KUKA KRL program: f1_Kuka_APT223T02S23.SRC

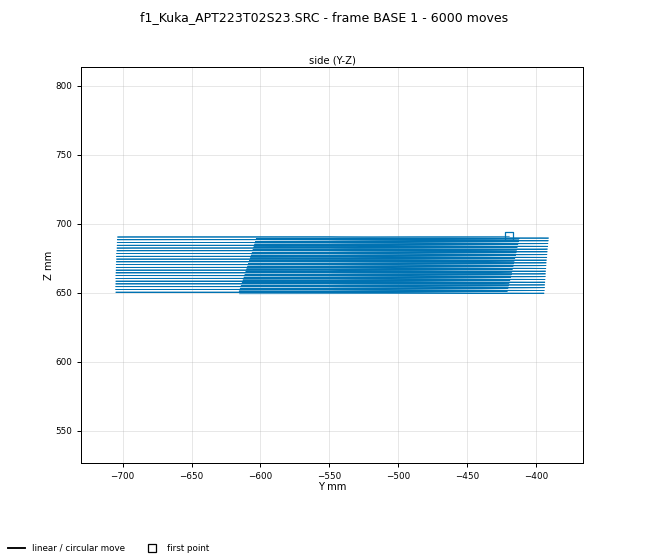
[picture p0: tool path of f1_Kuka_APT223T02S23.SRC in frame BASE 1, 6000 of 6001 moves have a stored position in this frame; points joined in program order, loops and branches not executed]
&ACCESS RVP
&REL 2
&PARAM TEMPLATE = C:\KRC\Roboter\Template\vorgabe
&PARAM EDITMASK = *
DEF f1_Kuka_APT223T02S23()


;FOLD INI;%{PE}%V3.2.0,%MKUKATPBASIS,%CINIT,%VCOMMON,%P
  ;FOLD BAS INI;%{E}%V3.2.0,%MKUKATPBASIS,%CINIT,%VINIT,%P
    GLOBAL INTERRUPT DECL 3 WHEN $STOPMESS==TRUE DO IR_STOPM ( )
    INTERRUPT ON 3
    BAS (#INITMOV,0 )
  ;ENDFOLD (BAS INI)
  ;FOLD USER INI;%{E}%V3.2.0,%MKUKATPUSER,%CINIT,%VINIT,%P
    ;Make your modifications here
  ;ENDFOLD (USER INI)
;ENDFOLD (INI)


;*** Make Null PTP Move
  PTP $pos_act

;*** Auto Load The Correct TOOL Data
  $tool=tool_data[2]

;*** Auto Load The Correct BASE Data
  $base=base_data[1]

  $ADVANCE = 5

;*** Restate Last Velocity
MMPM(30000.0)
SetRPM(8000)
LIN {X -0.177,Y -419.662,Z 690.937,A 0.000,B 0.000,C 90.000,E1 24.591} C_DIS
LIN {X 0.038,Y -422.624,Z 690.918,A 0.000,B 0.000,C 90.000,E1 21.173} C_DIS
LIN {X -0.096,Y -424.250,Z 690.908,A 0.000,B 0.000,C 90.000,E1 19.504} C_DIS
LIN {X -0.088,Y -425.859,Z 690.899,A 0.000,B 0.000,C 90.000,E1 17.819} C_DIS
LIN {X 0.034,Y -427.863,Z 690.888,A 0.000,B 0.000,C 90.000,E1 15.788} C_DIS
LIN {X -0.122,Y -430.468,Z 690.875,A 0.000,B 0.000,C 90.000,E1 13.467} C_DIS
LIN {X 0.099,Y -432.415,Z 690.866,A 0.000,B 0.000,C 90.000,E1 11.771} C_DIS
LIN {X -0.143,Y -434.451,Z 690.856,A 0.000,B 0.000,C 90.000,E1 10.141} C_DIS
LIN {X -0.149,Y -438.666,Z 690.838,A 0.000,B 0.000,C 90.000,E1 6.834} C_DIS
LIN {X -0.142,Y -441.750,Z 690.825,A 0.000,B 0.000,C 90.000,E1 4.531} C_DIS
LIN {X 0.024,Y -445.734,Z 690.811,A 0.000,B 0.000,C 90.000,E1 1.892} C_DIS
LIN {X -0.126,Y -449.793,Z 690.797,A 0.000,B 0.000,C 90.000,E1 359.484} C_DIS
LIN {X -0.170,Y -454.545,Z 690.783,A 0.000,B 0.000,C 90.000,E1 356.906} C_DIS
LIN {X 0.066,Y -458.306,Z 690.772,A 0.000,B 0.000,C 90.000,E1 354.951} C_DIS
LIN {X 0.178,Y -462.682,Z 690.760,A 0.000,B 0.000,C 90.000,E1 352.704} C_DIS
LIN {X -0.197,Y -466.311,Z 690.749,A 0.000,B 0.000,C 90.000,E1 350.849} C_DIS
LIN {X 0.236,Y -469.219,Z 690.740,A 0.000,B 0.000,C 90.000,E1 349.218} C_DIS
LIN {X 0.085,Y -472.585,Z 690.730,A 0.000,B 0.000,C 90.000,E1 347.353} C_DIS
LIN {X 0.213,Y -475.984,Z 690.719,A 0.000,B 0.000,C 90.000,E1 345.463} C_DIS
LIN {X 0.089,Y -479.488,Z 690.709,A 0.000,B 0.000,C 90.000,E1 343.614} C_DIS
LIN {X 0.195,Y -482.545,Z 690.701,A 0.000,B 0.000,C 90.000,E1 342.054} C_DIS
LIN {X 0.039,Y -484.409,Z 690.695,A 0.000,B 0.000,C 90.000,E1 341.148} C_DIS
LIN {X -0.067,Y -487.532,Z 690.687,A 0.000,B 0.000,C 90.000,E1 339.625} C_DIS
LIN {X -0.060,Y -491.876,Z 690.675,A 0.000,B 0.000,C 90.000,E1 337.486} C_DIS
LIN {X 0.051,Y -493.742,Z 690.670,A 0.000,B 0.000,C 90.000,E1 336.561} C_DIS
LIN {X -0.118,Y -495.162,Z 690.667,A 0.000,B 0.000,C 90.000,E1 335.973} C_DIS
LIN {X -0.024,Y -496.658,Z 690.663,A 0.000,B 0.000,C 90.000,E1 335.357} C_DIS
LIN {X -0.171,Y -498.186,Z 690.661,A 0.000,B 0.000,C 90.000,E1 334.921} C_DIS
LIN {X 0.097,Y -499.596,Z 690.659,A 0.000,B 0.000,C 90.000,E1 334.588} C_DIS
LIN {X -0.042,Y -501.612,Z 690.657,A 0.000,B 0.000,C 90.000,E1 334.280} C_DIS
LIN {X 0.069,Y -505.458,Z 690.655,A 0.000,B 0.000,C 90.000,E1 333.819} C_DIS
LIN {X -0.161,Y -510.103,Z 690.652,A 0.000,B 0.000,C 90.000,E1 333.435} C_DIS
LIN {X -0.285,Y -521.797,Z 690.648,A 0.000,B 0.000,C 90.000,E1 332.615} C_DIS
LIN {X -0.135,Y -531.169,Z 690.644,A 0.000,B 0.000,C 90.000,E1 331.975} C_DIS
LIN {X 0.252,Y -537.247,Z 690.642,A 0.000,B 0.000,C 90.000,E1 331.513} C_DIS
LIN {X 0.307,Y -541.703,Z 690.640,A 0.000,B 0.000,C 90.000,E1 331.179} C_DIS
LIN {X 0.113,Y -547.474,Z 690.638,A 0.000,B 0.000,C 90.000,E1 330.745} C_DIS
LIN {X 0.018,Y -553.101,Z 690.635,A 0.000,B 0.000,C 90.000,E1 330.284} C_DIS
LIN {X 0.032,Y -561.262,Z 690.631,A 0.000,B 0.000,C 90.000,E1 329.537} C_DIS
LIN {X -0.119,Y -571.528,Z 690.625,A 0.000,B 0.000,C 90.000,E1 328.535} C_DIS
LIN {X 0.210,Y -580.334,Z 690.620,A 0.000,B 0.000,C 90.000,E1 327.582} C_DIS
LIN {X -0.169,Y -591.315,Z 690.613,A 0.000,B 0.000,C 90.000,E1 326.421} C_DIS
LIN {X 0.068,Y -600.742,Z 690.608,A 0.000,B 0.000,C 90.000,E1 325.341} C_DIS
LIN {X 0.066,Y -605.196,Z 690.605,A 0.000,B 0.000,C 90.000,E1 324.815} C_DIS
LIN {X -0.294,Y -610.378,Z 690.601,A 0.000,B 0.000,C 90.000,E1 324.196} C_DIS
LIN {X 0.048,Y -617.140,Z 690.596,A 0.000,B 0.000,C 90.000,E1 323.256} C_DIS
LIN {X -0.223,Y -621.759,Z 690.592,A 0.000,B 0.000,C 90.000,E1 322.637} C_DIS
LIN {X 0.114,Y -629.358,Z 690.586,A 0.000,B 0.000,C 90.000,E1 321.457} C_DIS
LIN {X 0.322,Y -633.342,Z 690.582,A 0.000,B 0.000,C 90.000,E1 320.803} C_DIS
LIN {X 0.059,Y -637.842,Z 690.578,A 0.000,B 0.000,C 90.000,E1 320.070} C_DIS
LIN {X 0.157,Y -644.321,Z 690.572,A 0.000,B 0.000,C 90.000,E1 318.933} C_DIS
LIN {X 0.004,Y -647.101,Z 690.569,A 0.000,B 0.000,C 90.000,E1 318.447} C_DIS
LIN {X 0.242,Y -653.083,Z 690.563,A 0.000,B 0.000,C 90.000,E1 317.310} C_DIS
LIN {X 0.118,Y -656.784,Z 690.559,A 0.000,B 0.000,C 90.000,E1 316.581} C_DIS
LIN {X -0.428,Y -660.278,Z 690.555,A 0.000,B 0.000,C 90.000,E1 315.891} C_DIS
LIN {X -0.019,Y -663.506,Z 690.551,A 0.000,B 0.000,C 90.000,E1 315.121} C_DIS
LIN {X 0.423,Y -667.564,Z 690.545,A 0.000,B 0.000,C 90.000,E1 314.109} C_DIS
LIN {X -0.017,Y -671.440,Z 690.540,A 0.000,B 0.000,C 90.000,E1 313.176} C_DIS
LIN {X 0.069,Y -676.276,Z 690.533,A 0.000,B 0.000,C 90.000,E1 311.962} C_DIS
LIN {X -0.173,Y -680.748,Z 690.527,A 0.000,B 0.000,C 90.000,E1 310.782} C_DIS
LIN {X 0.106,Y -684.621,Z 690.520,A 0.000,B 0.000,C 90.000,E1 309.564} C_DIS
LIN {X 0.339,Y -686.758,Z 690.516,A 0.000,B 0.000,C 90.000,E1 308.830} C_DIS
LIN {X 0.221,Y -689.226,Z 690.511,A 0.000,B 0.000,C 90.000,E1 307.890} C_DIS
LIN {X 0.135,Y -691.500,Z 690.505,A 0.000,B 0.000,C 90.000,E1 306.950} C_DIS
LIN {X 0.073,Y -693.483,Z 690.500,A 0.000,B 0.000,C 90.000,E1 306.011} C_DIS
LIN {X -0.023,Y -694.830,Z 690.496,A 0.000,B 0.000,C 90.000,E1 305.311} C_DIS
LIN {X 0.245,Y -695.690,Z 690.494,A 0.000,B 0.000,C 90.000,E1 304.818} C_DIS
LIN {X -0.176,Y -697.121,Z 690.488,A 0.000,B 0.000,C 90.000,E1 303.913} C_DIS
LIN {X 0.344,Y -698.059,Z 690.484,A 0.000,B 0.000,C 90.000,E1 303.166} C_DIS
LIN {X -0.056,Y -699.136,Z 690.479,A 0.000,B 0.000,C 90.000,E1 302.260} C_DIS
LIN {X 0.061,Y -700.597,Z 690.471,A 0.000,B 0.000,C 90.000,E1 300.846} C_DIS
LIN {X 0.253,Y -701.115,Z 690.468,A 0.000,B 0.000,C 90.000,E1 300.129} C_DIS
LIN {X 0.050,Y -701.883,Z 690.460,A 0.000,B 0.000,C 90.000,E1 298.743} C_DIS
LIN {X 0.148,Y -702.599,Z 690.452,A 0.000,B 0.000,C 90.000,E1 297.334} C_DIS
LIN {X -0.078,Y -703.675,Z 690.443,A 0.000,B 0.000,C 90.000,E1 295.720} C_DIS
LIN {X -0.164,Y -703.404,Z 690.439,A 0.000,B 0.000,C 90.000,E1 295.027} C_DIS
LIN {X 0.399,Y -702.194,Z 690.436,A 0.000,B 0.000,C 90.000,E1 294.515} C_DIS
LIN {X -0.251,Y -701.369,Z 690.435,A 0.000,B 0.000,C 90.000,E1 294.335} C_DIS
LIN {X -0.113,Y -700.580,Z 690.435,A 0.000,B 0.000,C 90.000,E1 294.207} C_DIS
LIN {X 0.144,Y -696.444,Z 690.432,A 0.000,B 0.000,C 90.000,E1 293.718} C_DIS
LIN {X -0.363,Y -695.033,Z 690.431,A 0.000,B 0.000,C 90.000,E1 293.643} C_DIS
LIN {X -0.119,Y -692.958,Z 690.431,A 0.000,B 0.000,C 90.000,E1 293.515} C_DIS
LIN {X -0.070,Y -688.688,Z 690.430,A 0.000,B 0.000,C 90.000,E1 293.334} C_DIS
LIN {X -0.001,Y -684.521,Z 690.429,A 0.000,B 0.000,C 90.000,E1 293.206} C_DIS
LIN {X -0.212,Y -680.088,Z 690.428,A 0.000,B 0.000,C 90.000,E1 293.131} C_DIS
LIN {X 0.206,Y -675.238,Z 690.428,A 0.000,B 0.000,C 90.000,E1 293.025} C_DIS
LIN {X -0.219,Y -661.690,Z 690.427,A 0.000,B 0.000,C 90.000,E1 292.898} C_DIS
LIN {X -0.319,Y -644.942,Z 690.426,A 0.000,B 0.000,C 90.000,E1 292.642} C_DIS
LIN {X 0.098,Y -635.046,Z 690.425,A 0.000,B 0.000,C 90.000,E1 292.408} C_DIS
LIN {X 0.208,Y -621.578,Z 690.423,A 0.000,B 0.000,C 90.000,E1 292.078} C_DIS
LIN {X 0.164,Y -608.109,Z 690.421,A 0.000,B 0.000,C 90.000,E1 291.716} C_DIS
LIN {X -0.104,Y -576.806,Z 690.415,A 0.000,B 0.000,C 90.000,E1 290.791} C_DIS
LIN {X -0.048,Y -562.877,Z 690.413,A 0.000,B 0.000,C 90.000,E1 290.375} C_DIS
LIN {X -0.135,Y -558.097,Z 690.412,A 0.000,B 0.000,C 90.000,E1 290.174} C_DIS
LIN {X 0.037,Y -557.476,Z 690.412,A 0.000,B 0.000,C 90.000,E1 290.120} C_DIS
LIN {X -0.045,Y -555.543,Z 690.411,A 0.000,B 0.000,C 90.000,E1 289.939} C_DIS
LIN {X -0.085,Y -555.513,Z 690.411,A 0.000,B 0.000,C 90.000,E1 289.939} C_DIS
LIN {X -0.138,Y -554.733,Z 690.409,A 0.000,B 0.000,C 90.000,E1 289.631} C_DIS
LIN {X -0.156,Y -554.284,Z 690.407,A 0.000,B 0.000,C 90.000,E1 289.214} C_DIS
LIN {X 0.121,Y -553.763,Z 690.397,A 0.000,B 0.000,C 90.000,E1 287.511} C_DIS
LIN {X -0.066,Y -553.275,Z 690.390,A 0.000,B 0.000,C 90.000,E1 286.134} C_DIS
LIN {X 0.007,Y -552.908,Z 690.383,A 0.000,B 0.000,C 90.000,E1 285.009} C_DIS
LIN {X 0.194,Y -552.348,Z 690.376,A 0.000,B 0.000,C 90.000,E1 283.592} C_DIS
LIN {X -0.172,Y -551.606,Z 690.366,A 0.000,B 0.000,C 90.000,E1 281.951} C_DIS
LIN {X 0.098,Y -550.681,Z 690.355,A 0.000,B 0.000,C 90.000,E1 279.962} C_DIS
LIN {X -0.181,Y -549.760,Z 690.341,A 0.000,B 0.000,C 90.000,E1 277.466} C_DIS
LIN {X -0.056,Y -549.171,Z 690.326,A 0.000,B 0.000,C 90.000,E1 274.645} C_DIS
LIN {X 0.215,Y -549.047,Z 690.318,A 0.000,B 0.000,C 90.000,E1 273.212} C_DIS
LIN {X -0.105,Y -548.798,Z 690.312,A 0.000,B 0.000,C 90.000,E1 272.121} C_DIS
LIN {X 0.113,Y -548.447,Z 690.306,A 0.000,B 0.000,C 90.000,E1 270.974} C_DIS
LIN {X 0.263,Y -548.002,Z 690.301,A 0.000,B 0.000,C 90.000,E1 270.115} C_DIS
LIN {X -0.001,Y -547.042,Z 690.291,A 0.000,B 0.000,C 90.000,E1 268.453} C_DIS
LIN {X -0.210,Y -545.831,Z 690.281,A 0.000,B 0.000,C 90.000,E1 266.502} C_DIS
LIN {X 0.064,Y -544.611,Z 690.271,A 0.000,B 0.000,C 90.000,E1 264.780} C_DIS
LIN {X -0.203,Y -543.514,Z 690.263,A 0.000,B 0.000,C 90.000,E1 263.394} C_DIS
LIN {X 0.130,Y -541.476,Z 690.252,A 0.000,B 0.000,C 90.000,E1 261.376} C_DIS
LIN {X 0.172,Y -539.073,Z 690.238,A 0.000,B 0.000,C 90.000,E1 258.814} C_DIS
LIN {X -0.080,Y -538.081,Z 690.232,A 0.000,B 0.000,C 90.000,E1 257.701} C_DIS
LIN {X -0.160,Y -536.881,Z 690.224,A 0.000,B 0.000,C 90.000,E1 256.284} C_DIS
LIN {X 0.260,Y -535.598,Z 690.216,A 0.000,B 0.000,C 90.000,E1 254.810} C_DIS
LIN {X 0.273,Y -534.122,Z 690.208,A 0.000,B 0.000,C 90.000,E1 253.378} C_DIS
LIN {X -0.251,Y -532.665,Z 690.200,A 0.000,B 0.000,C 90.000,E1 252.000} C_DIS
LIN {X 0.059,Y -530.980,Z 690.190,A 0.000,B 0.000,C 90.000,E1 250.242} C_DIS
LIN {X -0.051,Y -529.919,Z 690.186,A 0.000,B 0.000,C 90.000,E1 249.390} C_DIS
LIN {X 0.057,Y -527.109,Z 690.174,A 0.000,B 0.000,C 90.000,E1 247.358} C_DIS
LIN {X -0.213,Y -525.432,Z 690.168,A 0.000,B 0.000,C 90.000,E1 246.230} C_DIS
LIN {X 0.033,Y -522.500,Z 690.158,A 0.000,B 0.000,C 90.000,E1 244.460} C_DIS
LIN {X 0.014,Y -520.939,Z 690.153,A 0.000,B 0.000,C 90.000,E1 243.589} C_DIS
LIN {X 0.112,Y -518.673,Z 690.147,A 0.000,B 0.000,C 90.000,E1 242.410} C_DIS
LIN {X -0.147,Y -515.816,Z 690.139,A 0.000,B 0.000,C 90.000,E1 240.973} C_DIS
LIN {X -0.023,Y -513.973,Z 690.134,A 0.000,B 0.000,C 90.000,E1 240.078} C_DIS
LIN {X -0.217,Y -510.196,Z 690.124,A 0.000,B 0.000,C 90.000,E1 238.329} C_DIS
LIN {X -0.114,Y -506.987,Z 690.116,A 0.000,B 0.000,C 90.000,E1 236.834} C_DIS
LIN {X 0.313,Y -504.278,Z 690.109,A 0.000,B 0.000,C 90.000,E1 235.595} C_DIS
LIN {X 0.168,Y -500.836,Z 690.101,A 0.000,B 0.000,C 90.000,E1 234.116} C_DIS
LIN {X 0.084,Y -497.917,Z 690.094,A 0.000,B 0.000,C 90.000,E1 232.924} C_DIS
LIN {X -0.138,Y -494.899,Z 690.087,A 0.000,B 0.000,C 90.000,E1 231.743} C_DIS
LIN {X -0.008,Y -490.504,Z 690.077,A 0.000,B 0.000,C 90.000,E1 229.908} C_DIS
LIN {X -0.075,Y -484.730,Z 690.064,A 0.000,B 0.000,C 90.000,E1 227.472} C_DIS
LIN {X -0.011,Y -479.137,Z 690.050,A 0.000,B 0.000,C 90.000,E1 225.000} C_DIS
LIN {X -0.104,Y -475.497,Z 690.041,A 0.000,B 0.000,C 90.000,E1 223.461} C_DIS
LIN {X -0.072,Y -470.576,Z 690.029,A 0.000,B 0.000,C 90.000,E1 221.272} C_DIS
LIN {X -0.258,Y -467.231,Z 690.021,A 0.000,B 0.000,C 90.000,E1 219.725} C_DIS
LIN {X 0.155,Y -463.901,Z 690.012,A 0.000,B 0.000,C 90.000,E1 218.096} C_DIS
LIN {X 0.034,Y -457.033,Z 689.992,A 0.000,B 0.000,C 90.000,E1 214.612} C_DIS
LIN {X -0.296,Y -454.541,Z 689.985,A 0.000,B 0.000,C 90.000,E1 213.372} C_DIS
LIN {X 0.140,Y -450.873,Z 689.974,A 0.000,B 0.000,C 90.000,E1 211.386} C_DIS
LIN {X -0.134,Y -446.600,Z 689.962,A 0.000,B 0.000,C 90.000,E1 209.155} C_DIS
LIN {X 0.027,Y -443.112,Z 689.951,A 0.000,B 0.000,C 90.000,E1 207.180} C_DIS
LIN {X 0.083,Y -439.517,Z 689.940,A 0.000,B 0.000,C 90.000,E1 205.207} C_DIS
LIN {X 0.027,Y -437.117,Z 689.933,A 0.000,B 0.000,C 90.000,E1 203.898} C_DIS
LIN {X 0.162,Y -433.497,Z 689.922,A 0.000,B 0.000,C 90.000,E1 201.897} C_DIS
LIN {X 0.072,Y -430.490,Z 689.913,A 0.000,B 0.000,C 90.000,E1 200.248} C_DIS
LIN {X 0.126,Y -426.762,Z 689.901,A 0.000,B 0.000,C 90.000,E1 198.236} C_DIS
LIN {X 0.010,Y -422.649,Z 689.888,A 0.000,B 0.000,C 90.000,E1 195.898} C_DIS
LIN {X 0.147,Y -419.745,Z 689.879,A 0.000,B 0.000,C 90.000,E1 194.189} C_DIS
LIN {X 0.069,Y -415.050,Z 689.864,A 0.000,B 0.000,C 90.000,E1 191.478} C_DIS
LIN {X -0.068,Y -411.729,Z 689.852,A 0.000,B 0.000,C 90.000,E1 189.443} C_DIS
LIN {X 0.094,Y -409.036,Z 689.843,A 0.000,B 0.000,C 90.000,E1 187.701} C_DIS
LIN {X 0.135,Y -406.468,Z 689.833,A 0.000,B 0.000,C 90.000,E1 185.967} C_DIS
LIN {X 0.002,Y -403.075,Z 689.820,A 0.000,B 0.000,C 90.000,E1 183.555} C_DIS
LIN {X 0.159,Y -400.088,Z 689.806,A 0.000,B 0.000,C 90.000,E1 181.088} C_DIS
LIN {X 0.110,Y -396.926,Z 689.789,A 0.000,B 0.000,C 90.000,E1 177.936} C_DIS
LIN {X 0.061,Y -394.730,Z 689.773,A 0.000,B 0.000,C 90.000,E1 175.122} C_DIS
LIN {X -0.117,Y -392.750,Z 689.751,A 0.000,B 0.000,C 90.000,E1 171.254} C_DIS
LIN {X -0.029,Y -392.123,Z 689.738,A 0.000,B 0.000,C 90.000,E1 168.757} C_DIS
LIN {X -0.101,Y -391.771,Z 689.728,A 0.000,B 0.000,C 90.000,E1 166.992} C_DIS
LIN {X -0.064,Y -391.172,Z 689.708,A 0.000,B 0.000,C 90.000,E1 163.433} C_DIS
LIN {X 0.188,Y -391.169,Z 689.692,A 0.000,B 0.000,C 90.000,E1 160.550} C_DIS
LIN {X 0.091,Y -391.330,Z 689.676,A 0.000,B 0.000,C 90.000,E1 157.720} C_DIS
LIN {X -0.089,Y -391.469,Z 689.664,A 0.000,B 0.000,C 90.000,E1 155.613} C_DIS
LIN {X -0.106,Y -391.736,Z 689.651,A 0.000,B 0.000,C 90.000,E1 153.127} C_DIS
LIN {X 0.105,Y -392.346,Z 689.635,A 0.000,B 0.000,C 90.000,E1 150.255} C_DIS
LIN {X -0.010,Y -393.124,Z 689.621,A 0.000,B 0.000,C 90.000,E1 147.788} C_DIS
LIN {X -0.212,Y -394.831,Z 689.601,A 0.000,B 0.000,C 90.000,E1 144.276} C_DIS
LIN {X 0.012,Y -396.062,Z 689.592,A 0.000,B 0.000,C 90.000,E1 142.477} C_DIS
LIN {X 0.158,Y -398.083,Z 689.578,A 0.000,B 0.000,C 90.000,E1 139.989} C_DIS
LIN {X 0.086,Y -399.704,Z 689.568,A 0.000,B 0.000,C 90.000,E1 138.243} C_DIS
LIN {X -0.047,Y -402.173,Z 689.555,A 0.000,B 0.000,C 90.000,E1 135.810} C_DIS
LIN {X 0.082,Y -403.736,Z 689.550,A 0.000,B 0.000,C 90.000,E1 134.919} C_DIS
LIN {X 0.078,Y -405.791,Z 689.546,A 0.000,B 0.000,C 90.000,E1 134.190} C_DIS
LIN {X -0.089,Y -407.601,Z 689.544,A 0.000,B 0.000,C 90.000,E1 133.866} C_DIS
LIN {X -0.210,Y -408.808,Z 689.542,A 0.000,B 0.000,C 90.000,E1 133.623} C_DIS
LIN {X -0.029,Y -410.740,Z 689.541,A 0.000,B 0.000,C 90.000,E1 133.338} C_DIS
LIN {X -0.106,Y -411.886,Z 689.540,A 0.000,B 0.000,C 90.000,E1 133.176} C_DIS
LIN {X -0.197,Y -416.632,Z 689.537,A 0.000,B 0.000,C 90.000,E1 132.690} C_DIS
LIN {X -0.118,Y -433.549,Z 689.529,A 0.000,B 0.000,C 90.000,E1 131.148} C_DIS
LIN {X 0.013,Y -448.902,Z 689.521,A 0.000,B 0.000,C 90.000,E1 129.850} C_DIS
LIN {X -0.164,Y -462.908,Z 689.515,A 0.000,B 0.000,C 90.000,E1 128.749} C_DIS
LIN {X 0.034,Y -468.842,Z 689.512,A 0.000,B 0.000,C 90.000,E1 128.222} C_DIS
LIN {X 0.051,Y -477.755,Z 689.508,A 0.000,B 0.000,C 90.000,E1 127.443} C_DIS
LIN {X -0.050,Y -484.911,Z 689.504,A 0.000,B 0.000,C 90.000,E1 126.790} C_DIS
LIN {X 0.072,Y -493.460,Z 689.500,A 0.000,B 0.000,C 90.000,E1 125.964} C_DIS
LIN {X -0.144,Y -498.944,Z 689.497,A 0.000,B 0.000,C 90.000,E1 125.438} C_DIS
LIN {X -0.289,Y -504.315,Z 689.494,A 0.000,B 0.000,C 90.000,E1 124.898} C_DIS
LIN {X -0.281,Y -507.046,Z 689.492,A 0.000,B 0.000,C 90.000,E1 124.612} C_DIS
LIN {X -0.129,Y -513.089,Z 689.488,A 0.000,B 0.000,C 90.000,E1 123.913} C_DIS
LIN {X -0.188,Y -516.672,Z 689.486,A 0.000,B 0.000,C 90.000,E1 123.499} C_DIS
LIN {X -0.176,Y -521.024,Z 689.483,A 0.000,B 0.000,C 90.000,E1 122.959} C_DIS
LIN {X -0.188,Y -525.187,Z 689.480,A 0.000,B 0.000,C 90.000,E1 122.418} C_DIS
LIN {X 0.169,Y -529.277,Z 689.477,A 0.000,B 0.000,C 90.000,E1 121.799} C_DIS
LIN {X 0.035,Y -533.666,Z 689.473,A 0.000,B 0.000,C 90.000,E1 121.131} C_DIS
LIN {X -0.162,Y -537.023,Z 689.470,A 0.000,B 0.000,C 90.000,E1 120.590} C_DIS
LIN {X -0.260,Y -541.499,Z 689.465,A 0.000,B 0.000,C 90.000,E1 119.745} C_DIS
LIN {X 0.085,Y -544.958,Z 689.461,A 0.000,B 0.000,C 90.000,E1 118.999} C_DIS
LIN {X 0.075,Y -548.802,Z 689.456,A 0.000,B 0.000,C 90.000,E1 118.153} C_DIS
LIN {X 0.083,Y -551.249,Z 689.453,A 0.000,B 0.000,C 90.000,E1 117.590} C_DIS
LIN {X 0.139,Y -554.580,Z 689.449,A 0.000,B 0.000,C 90.000,E1 116.744} C_DIS
LIN {X 0.006,Y -558.705,Z 689.443,A 0.000,B 0.000,C 90.000,E1 115.643} C_DIS
LIN {X -0.115,Y -561.579,Z 689.438,A 0.000,B 0.000,C 90.000,E1 114.823} C_DIS
LIN {X 0.309,Y -564.176,Z 689.433,A 0.000,B 0.000,C 90.000,E1 113.951} C_DIS
LIN {X 0.024,Y -566.557,Z 689.429,A 0.000,B 0.000,C 90.000,E1 113.153} C_DIS
LIN {X -0.014,Y -568.549,Z 689.424,A 0.000,B 0.000,C 90.000,E1 112.333} C_DIS
LIN {X -0.081,Y -571.418,Z 689.417,A 0.000,B 0.000,C 90.000,E1 110.972} C_DIS
LIN {X 0.247,Y -572.998,Z 689.412,A 0.000,B 0.000,C 90.000,E1 110.120} C_DIS
LIN {X -0.313,Y -575.878,Z 689.403,A 0.000,B 0.000,C 90.000,E1 108.544} C_DIS
LIN {X 0.078,Y -578.303,Z 689.395,A 0.000,B 0.000,C 90.000,E1 107.149} C_DIS
LIN {X 0.176,Y -580.646,Z 689.388,A 0.000,B 0.000,C 90.000,E1 105.788} C_DIS
LIN {X 0.098,Y -582.456,Z 689.382,A 0.000,B 0.000,C 90.000,E1 104.717} C_DIS
LIN {X 0.276,Y -584.612,Z 689.374,A 0.000,B 0.000,C 90.000,E1 103.355} C_DIS
LIN {X 0.034,Y -587.176,Z 689.365,A 0.000,B 0.000,C 90.000,E1 101.771} C_DIS
LIN {X -0.105,Y -588.958,Z 689.359,A 0.000,B 0.000,C 90.000,E1 100.715} C_DIS
LIN {X -0.067,Y -591.044,Z 689.352,A 0.000,B 0.000,C 90.000,E1 99.378} C_DIS
LIN {X 0.319,Y -592.602,Z 689.346,A 0.000,B 0.000,C 90.000,E1 98.276} C_DIS
LIN {X -0.059,Y -594.789,Z 689.337,A 0.000,B 0.000,C 90.000,E1 96.720} C_DIS
LIN {X 0.205,Y -596.779,Z 689.329,A 0.000,B 0.000,C 90.000,E1 95.106} C_DIS
LIN {X 0.227,Y -598.397,Z 689.321,A 0.000,B 0.000,C 90.000,E1 93.784} C_DIS
LIN {X 0.000,Y -599.516,Z 689.315,A 0.000,B 0.000,C 90.000,E1 92.751} C_DIS
LIN {X -0.217,Y -600.462,Z 689.310,A 0.000,B 0.000,C 90.000,E1 91.718} C_DIS
LIN {X 0.163,Y -601.305,Z 689.304,A 0.000,B 0.000,C 90.000,E1 90.630} C_DIS
LIN {X -0.042,Y -601.948,Z 689.298,A 0.000,B 0.000,C 90.000,E1 89.599} C_DIS
LIN {X 0.280,Y -602.580,Z 689.289,A 0.000,B 0.000,C 90.000,E1 87.993} C_DIS
LIN {X 0.081,Y -602.864,Z 689.283,A 0.000,B 0.000,C 90.000,E1 86.963} C_DIS
LIN {X -0.156,Y -603.080,Z 689.274,A 0.000,B 0.000,C 90.000,E1 85.412} C_DIS
LIN {X -0.274,Y -603.046,Z 689.269,A 0.000,B 0.000,C 90.000,E1 84.375} C_DIS
LIN {X 0.211,Y -602.874,Z 689.263,A 0.000,B 0.000,C 90.000,E1 83.280} C_DIS
LIN {X 0.092,Y -602.603,Z 689.257,A 0.000,B 0.000,C 90.000,E1 82.243} C_DIS
LIN {X 0.050,Y -602.232,Z 689.251,A 0.000,B 0.000,C 90.000,E1 81.197} C_DIS
LIN {X 0.008,Y -601.520,Z 689.245,A 0.000,B 0.000,C 90.000,E1 80.151} C_DIS
LIN {X 0.259,Y -600.418,Z 689.238,A 0.000,B 0.000,C 90.000,E1 78.814} C_DIS
LIN {X 0.020,Y -599.157,Z 689.231,A 0.000,B 0.000,C 90.000,E1 77.521} C_DIS
LIN {X -0.237,Y -597.751,Z 689.223,A 0.000,B 0.000,C 90.000,E1 76.228} C_DIS
LIN {X -0.087,Y -595.949,Z 689.215,A 0.000,B 0.000,C 90.000,E1 74.629} C_DIS
LIN {X -0.257,Y -594.253,Z 689.207,A 0.000,B 0.000,C 90.000,E1 73.323} C_DIS
LIN {X -0.289,Y -592.447,Z 689.200,A 0.000,B 0.000,C 90.000,E1 72.000} C_DIS
LIN {X -0.038,Y -590.843,Z 689.194,A 0.000,B 0.000,C 90.000,E1 70.913} C_DIS
LIN {X 0.061,Y -588.608,Z 689.187,A 0.000,B 0.000,C 90.000,E1 69.571} C_DIS
LIN {X -0.090,Y -586.633,Z 689.181,A 0.000,B 0.000,C 90.000,E1 68.518} C_DIS
LIN {X 0.279,Y -584.452,Z 689.175,A 0.000,B 0.000,C 90.000,E1 67.411} C_DIS
LIN {X 0.071,Y -581.946,Z 689.169,A 0.000,B 0.000,C 90.000,E1 66.357} C_DIS
LIN {X 0.063,Y -579.109,Z 689.163,A 0.000,B 0.000,C 90.000,E1 65.281} C_DIS
LIN {X 0.164,Y -576.819,Z 689.158,A 0.000,B 0.000,C 90.000,E1 64.460} C_DIS
LIN {X 0.237,Y -574.314,Z 689.154,A 0.000,B 0.000,C 90.000,E1 63.640} C_DIS
LIN {X 0.114,Y -570.746,Z 689.148,A 0.000,B 0.000,C 90.000,E1 62.564} C_DIS
LIN {X -0.303,Y -566.780,Z 689.142,A 0.000,B 0.000,C 90.000,E1 61.513} C_DIS
LIN {X 0.104,Y -564.705,Z 689.139,A 0.000,B 0.000,C 90.000,E1 60.923} C_DIS
LIN {X -0.189,Y -561.238,Z 689.134,A 0.000,B 0.000,C 90.000,E1 60.127} C_DIS
LIN {X 0.175,Y -558.793,Z 689.131,A 0.000,B 0.000,C 90.000,E1 59.537} C_DIS
LIN {X -0.064,Y -555.258,Z 689.127,A 0.000,B 0.000,C 90.000,E1 58.869} C_DIS
LIN {X -0.227,Y -551.404,Z 689.123,A 0.000,B 0.000,C 90.000,E1 58.201} C_DIS
LIN {X 0.219,Y -547.011,Z 689.119,A 0.000,B 0.000,C 90.000,E1 57.454} C_DIS
LIN {X -0.003,Y -543.251,Z 689.116,A 0.000,B 0.000,C 90.000,E1 56.914} C_DIS
LIN {X -0.109,Y -540.094,Z 689.114,A 0.000,B 0.000,C 90.000,E1 56.501} C_DIS
LIN {X 0.050,Y -539.087,Z 689.113,A 0.000,B 0.000,C 90.000,E1 56.342} C_DIS
LIN {X -0.223,Y -534.455,Z 689.110,A 0.000,B 0.000,C 90.000,E1 55.801} C_DIS
LIN {X 0.304,Y -529.243,Z 689.107,A 0.000,B 0.000,C 90.000,E1 55.182} C_DIS
LIN {X -0.031,Y -525.146,Z 689.105,A 0.000,B 0.000,C 90.000,E1 54.815} C_DIS
LIN {X -0.133,Y -519.437,Z 689.102,A 0.000,B 0.000,C 90.000,E1 54.322} C_DIS
LIN {X 0.128,Y -513.470,Z 689.099,A 0.000,B 0.000,C 90.000,E1 53.829} C_DIS
LIN {X -0.007,Y -508.636,Z 689.097,A 0.000,B 0.000,C 90.000,E1 53.497} C_DIS
LIN {X 0.004,Y -500.368,Z 689.094,A 0.000,B 0.000,C 90.000,E1 52.970} C_DIS
LIN {X -0.027,Y -492.109,Z 689.092,A 0.000,B 0.000,C 90.000,E1 52.477} C_DIS
LIN {X -0.022,Y -475.500,Z 689.086,A 0.000,B 0.000,C 90.000,E1 51.537} C_DIS
LIN {X 0.040,Y -453.997,Z 689.079,A 0.000,B 0.000,C 90.000,E1 50.275} C_DIS
LIN {X -0.056,Y -435.964,Z 689.073,A 0.000,B 0.000,C 90.000,E1 49.175} C_DIS
LIN {X -0.092,Y -428.102,Z 689.070,A 0.000,B 0.000,C 90.000,E1 48.647} C_DIS
LIN {X -0.148,Y -425.824,Z 689.069,A 0.000,B 0.000,C 90.000,E1 48.485} C_DIS
LIN {X -0.172,Y -425.813,Z 689.069,A 0.000,B 0.000,C 90.000,E1 48.485} C_DIS
LIN {X 0.028,Y -418.406,Z 689.049,A 0.000,B 0.000,C 90.000,E1 44.717} C_DIS
LIN {X 0.004,Y -412.583,Z 689.034,A 0.000,B 0.000,C 90.000,E1 42.162} C_DIS
LIN {X 0.177,Y -412.612,Z 689.020,A 0.000,B 0.000,C 90.000,E1 39.564} C_DIS
LIN {X -0.024,Y -413.406,Z 689.003,A 0.000,B 0.000,C 90.000,E1 36.503} C_DIS
LIN {X 0.175,Y -414.027,Z 688.995,A 0.000,B 0.000,C 90.000,E1 35.105} C_DIS
LIN {X -0.082,Y -414.995,Z 688.984,A 0.000,B 0.000,C 90.000,E1 33.086} C_DIS
LIN {X -0.146,Y -415.948,Z 688.974,A 0.000,B 0.000,C 90.000,E1 31.386} C_DIS
LIN {X -0.104,Y -417.041,Z 688.963,A 0.000,B 0.000,C 90.000,E1 29.333} C_DIS
LIN {X 0.130,Y -418.272,Z 688.952,A 0.000,B 0.000,C 90.000,E1 27.257} C_DIS
LIN {X -0.027,Y -419.925,Z 688.938,A 0.000,B 0.000,C 90.000,E1 24.899} C_DIS
LIN {X -0.198,Y -422.822,Z 688.920,A 0.000,B 0.000,C 90.000,E1 21.535} C_DIS
LIN {X 0.069,Y -424.449,Z 688.910,A 0.000,B 0.000,C 90.000,E1 19.812} C_DIS
LIN {X 0.084,Y -426.031,Z 688.901,A 0.000,B 0.000,C 90.000,E1 18.127} C_DIS
LIN {X -0.075,Y -427.971,Z 688.890,A 0.000,B 0.000,C 90.000,E1 16.134} C_DIS
LIN {X -0.024,Y -430.051,Z 688.878,A 0.000,B 0.000,C 90.000,E1 14.120} C_DIS
LIN {X -0.230,Y -432.004,Z 688.869,A 0.000,B 0.000,C 90.000,E1 12.479} C_DIS
LIN {X -0.143,Y -434.753,Z 688.856,A 0.000,B 0.000,C 90.000,E1 10.141} C_DIS
LIN {X -0.137,Y -438.930,Z 688.838,A 0.000,B 0.000,C 90.000,E1 6.834} C_DIS
LIN {X -0.123,Y -442.003,Z 688.825,A 0.000,B 0.000,C 90.000,E1 4.531} C_DIS
LIN {X -0.085,Y -445.447,Z 688.812,A 0.000,B 0.000,C 90.000,E1 2.236} C_DIS
LIN {X 0.170,Y -449.453,Z 688.799,A 0.000,B 0.000,C 90.000,E1 359.771} C_DIS
LIN {X -0.163,Y -454.746,Z 688.783,A 0.000,B 0.000,C 90.000,E1 356.906} C_DIS
LIN {X 0.077,Y -458.474,Z 688.772,A 0.000,B 0.000,C 90.000,E1 354.951} C_DIS
LIN {X 0.194,Y -462.819,Z 688.760,A 0.000,B 0.000,C 90.000,E1 352.704} C_DIS
LIN {X -0.178,Y -466.439,Z 688.749,A 0.000,B 0.000,C 90.000,E1 350.849} C_DIS
LIN {X 0.258,Y -469.348,Z 688.740,A 0.000,B 0.000,C 90.000,E1 349.218} C_DIS
LIN {X 0.109,Y -472.697,Z 688.730,A 0.000,B 0.000,C 90.000,E1 347.353} C_DIS
LIN {X 0.076,Y -476.665,Z 688.718,A 0.000,B 0.000,C 90.000,E1 345.172} C_DIS
LIN {X -0.040,Y -480.191,Z 688.707,A 0.000,B 0.000,C 90.000,E1 343.323} C_DIS
LIN {X 0.227,Y -482.643,Z 688.701,A 0.000,B 0.000,C 90.000,E1 342.054} C_DIS
LIN {X -0.081,Y -485.110,Z 688.694,A 0.000,B 0.000,C 90.000,E1 340.859} C_DIS
LIN {X -0.032,Y -487.633,Z 688.687,A 0.000,B 0.000,C 90.000,E1 339.625} C_DIS
LIN {X -0.055,Y -491.348,Z 688.677,A 0.000,B 0.000,C 90.000,E1 337.794} C_DIS
LIN {X -0.078,Y -495.085,Z 688.667,A 0.000,B 0.000,C 90.000,E1 335.973} C_DIS
LIN {X 0.016,Y -496.497,Z 688.663,A 0.000,B 0.000,C 90.000,E1 335.357} C_DIS
LIN {X 0.328,Y -498.265,Z 688.660,A 0.000,B 0.000,C 90.000,E1 334.717} C_DIS
LIN {X 0.188,Y -500.243,Z 688.657,A 0.000,B 0.000,C 90.000,E1 334.280} C_DIS
LIN {X 0.055,Y -503.276,Z 688.655,A 0.000,B 0.000,C 90.000,E1 333.845} C_DIS
LIN {X 0.071,Y -506.248,Z 688.653,A 0.000,B 0.000,C 90.000,E1 333.512} C_DIS
LIN {X -0.148,Y -510.833,Z 688.651,A 0.000,B 0.000,C 90.000,E1 333.127} C_DIS
LIN {X -0.177,Y -522.806,Z 688.646,A 0.000,B 0.000,C 90.000,E1 332.281} C_DIS
LIN {X 0.209,Y -533.705,Z 688.642,A 0.000,B 0.000,C 90.000,E1 331.513} C_DIS
LIN {X -0.196,Y -539.736,Z 688.640,A 0.000,B 0.000,C 90.000,E1 331.129} C_DIS
LIN {X -0.052,Y -545.503,Z 688.637,A 0.000,B 0.000,C 90.000,E1 330.667} C_DIS
LIN {X -0.121,Y -551.160,Z 688.634,A 0.000,B 0.000,C 90.000,E1 330.205} C_DIS
LIN {X -0.071,Y -556.685,Z 688.632,A 0.000,B 0.000,C 90.000,E1 329.715} C_DIS
LIN {X 0.021,Y -562.029,Z 688.629,A 0.000,B 0.000,C 90.000,E1 329.203} C_DIS
LIN {X -0.231,Y -569.912,Z 688.625,A 0.000,B 0.000,C 90.000,E1 328.456} C_DIS
LIN {X -0.123,Y -577.555,Z 688.620,A 0.000,B 0.000,C 90.000,E1 327.661} C_DIS
LIN {X 0.001,Y -587.430,Z 688.614,A 0.000,B 0.000,C 90.000,E1 326.580} C_DIS
LIN {X -0.115,Y -593.498,Z 688.611,A 0.000,B 0.000,C 90.000,E1 325.928} C_DIS
LIN {X 0.166,Y -601.794,Z 688.606,A 0.000,B 0.000,C 90.000,E1 324.975} C_DIS
LIN {X -0.175,Y -606.174,Z 688.603,A 0.000,B 0.000,C 90.000,E1 324.482} C_DIS
LIN {X -0.173,Y -611.283,Z 688.599,A 0.000,B 0.000,C 90.000,E1 323.829} C_DIS
LIN {X 0.006,Y -617.055,Z 688.595,A 0.000,B 0.000,C 90.000,E1 323.050} C_DIS
LIN {X 0.082,Y -622.520,Z 688.591,A 0.000,B 0.000,C 90.000,E1 322.271} C_DIS
LIN {X 0.062,Y -629.311,Z 688.585,A 0.000,B 0.000,C 90.000,E1 321.251} C_DIS
LIN {X -0.240,Y -634.081,Z 688.581,A 0.000,B 0.000,C 90.000,E1 320.517} C_DIS
LIN {X 0.202,Y -641.481,Z 688.574,A 0.000,B 0.000,C 90.000,E1 319.218} C_DIS
LIN {X -0.053,Y -646.400,Z 688.569,A 0.000,B 0.000,C 90.000,E1 318.366} C_DIS
LIN {X -0.259,Y -651.831,Z 688.563,A 0.000,B 0.000,C 90.000,E1 317.391} C_DIS
LIN {X 0.077,Y -655.597,Z 688.559,A 0.000,B 0.000,C 90.000,E1 316.620} C_DIS
LIN {X 0.455,Y -658.611,Z 688.556,A 0.000,B 0.000,C 90.000,E1 315.972} C_DIS
LIN {X -0.084,Y -661.978,Z 688.552,A 0.000,B 0.000,C 90.000,E1 315.283} C_DIS
LIN {X 0.335,Y -666.120,Z 688.546,A 0.000,B 0.000,C 90.000,E1 314.271} C_DIS
LIN {X -0.114,Y -671.110,Z 688.539,A 0.000,B 0.000,C 90.000,E1 313.095} C_DIS
LIN {X -0.036,Y -676.025,Z 688.533,A 0.000,B 0.000,C 90.000,E1 311.881} C_DIS
LIN {X -0.283,Y -680.531,Z 688.526,A 0.000,B 0.000,C 90.000,E1 310.701} C_DIS
LIN {X -0.010,Y -684.463,Z 688.519,A 0.000,B 0.000,C 90.000,E1 309.483} C_DIS
LIN {X -0.162,Y -687.226,Z 688.514,A 0.000,B 0.000,C 90.000,E1 308.543} C_DIS
LIN {X -0.274,Y -689.738,Z 688.509,A 0.000,B 0.000,C 90.000,E1 307.604} C_DIS
LIN {X -0.356,Y -691.947,Z 688.504,A 0.000,B 0.000,C 90.000,E1 306.664} C_DIS
LIN {X -0.058,Y -693.455,Z 688.500,A 0.000,B 0.000,C 90.000,E1 305.931} C_DIS
LIN {X 0.062,Y -695.239,Z 688.494,A 0.000,B 0.000,C 90.000,E1 304.978} C_DIS
LIN {X 0.032,Y -696.795,Z 688.489,A 0.000,B 0.000,C 90.000,E1 304.040} C_DIS
LIN {X -0.421,Y -697.789,Z 688.485,A 0.000,B 0.000,C 90.000,E1 303.372} C_DIS
LIN {X 0.051,Y -699.422,Z 688.477,A 0.000,B 0.000,C 90.000,E1 301.926} C_DIS
LIN {X -0.110,Y -700.463,Z 688.472,A 0.000,B 0.000,C 90.000,E1 301.003} C_DIS
LIN {X 0.101,Y -701.165,Z 688.467,A 0.000,B 0.000,C 90.000,E1 300.050} C_DIS
LIN {X 0.234,Y -701.855,Z 688.461,A 0.000,B 0.000,C 90.000,E1 298.871} C_DIS
LIN {X -0.294,Y -702.599,Z 688.453,A 0.000,B 0.000,C 90.000,E1 297.513} C_DIS
LIN {X 0.105,Y -703.678,Z 688.444,A 0.000,B 0.000,C 90.000,E1 295.848} C_DIS
LIN {X 0.388,Y -703.795,Z 688.442,A 0.000,B 0.000,C 90.000,E1 295.591} C_DIS
LIN {X 0.019,Y -703.605,Z 688.440,A 0.000,B 0.000,C 90.000,E1 295.155} C_DIS
LIN {X 0.302,Y -703.265,Z 688.439,A 0.000,B 0.000,C 90.000,E1 294.899} C_DIS
LIN {X -0.065,Y -701.943,Z 688.436,A 0.000,B 0.000,C 90.000,E1 294.463} C_DIS
LIN {X 0.213,Y -700.770,Z 688.435,A 0.000,B 0.000,C 90.000,E1 294.207} C_DIS
LIN {X -0.169,Y -696.531,Z 688.432,A 0.000,B 0.000,C 90.000,E1 293.770} C_DIS
LIN {X -0.039,Y -695.197,Z 688.431,A 0.000,B 0.000,C 90.000,E1 293.643} C_DIS
LIN {X 0.089,Y -693.090,Z 688.431,A 0.000,B 0.000,C 90.000,E1 293.515} C_DIS
LIN {X 0.211,Y -688.895,Z 688.430,A 0.000,B 0.000,C 90.000,E1 293.334} C_DIS
LIN {X 0.128,Y -684.192,Z 688.429,A 0.000,B 0.000,C 90.000,E1 293.206} C_DIS
LIN {X -0.082,Y -679.654,Z 688.429,A 0.000,B 0.000,C 90.000,E1 293.131} C_DIS
LIN {X -0.199,Y -670.738,Z 688.428,A 0.000,B 0.000,C 90.000,E1 293.025} C_DIS
LIN {X -0.257,Y -659.941,Z 688.427,A 0.000,B 0.000,C 90.000,E1 292.898} C_DIS
LIN {X 0.196,Y -646.379,Z 688.426,A 0.000,B 0.000,C 90.000,E1 292.642} C_DIS
LIN {X 0.052,Y -636.188,Z 688.425,A 0.000,B 0.000,C 90.000,E1 292.461} C_DIS
LIN {X -0.131,Y -619.557,Z 688.423,A 0.000,B 0.000,C 90.000,E1 292.078} C_DIS
LIN {X -0.254,Y -606.101,Z 688.421,A 0.000,B 0.000,C 90.000,E1 291.716} C_DIS
LIN {X -0.013,Y -576.446,Z 688.416,A 0.000,B 0.000,C 90.000,E1 290.791} C_DIS
LIN {X 0.041,Y -562.486,Z 688.413,A 0.000,B 0.000,C 90.000,E1 290.375} C_DIS
LIN {X 0.295,Y -557.451,Z 688.412,A 0.000,B 0.000,C 90.000,E1 290.120} C_DIS
LIN {X 0.278,Y -555.572,Z 688.411,A 0.000,B 0.000,C 90.000,E1 289.939} C_DIS
LIN {X 0.239,Y -555.552,Z 688.411,A 0.000,B 0.000,C 90.000,E1 289.939} C_DIS
LIN {X 0.097,Y -554.779,Z 688.409,A 0.000,B 0.000,C 90.000,E1 289.685} C_DIS
LIN {X 0.158,Y -554.218,Z 688.406,A 0.000,B 0.000,C 90.000,E1 289.087} C_DIS
LIN {X 0.154,Y -553.823,Z 688.398,A 0.000,B 0.000,C 90.000,E1 287.692} C_DIS
LIN {X -0.031,Y -553.344,Z 688.391,A 0.000,B 0.000,C 90.000,E1 286.315} C_DIS
LIN {X 0.044,Y -552.995,Z 688.384,A 0.000,B 0.000,C 90.000,E1 285.190} C_DIS
LIN {X 0.235,Y -552.430,Z 688.377,A 0.000,B 0.000,C 90.000,E1 283.772} C_DIS
LIN {X -0.010,Y -551.677,Z 688.367,A 0.000,B 0.000,C 90.000,E1 282.119} C_DIS
LIN {X 0.155,Y -550.743,Z 688.357,A 0.000,B 0.000,C 90.000,E1 280.141} C_DIS
LIN {X -0.109,Y -549.801,Z 688.342,A 0.000,B 0.000,C 90.000,E1 277.644} C_DIS
LIN {X 0.124,Y -549.201,Z 688.325,A 0.000,B 0.000,C 90.000,E1 274.531} C_DIS
LIN {X -0.150,Y -549.071,Z 688.318,A 0.000,B 0.000,C 90.000,E1 273.154} C_DIS
LIN {X 0.079,Y -548.796,Z 688.311,A 0.000,B 0.000,C 90.000,E1 272.007} C_DIS
LIN {X -0.251,Y -548.436,Z 688.305,A 0.000,B 0.000,C 90.000,E1 270.917} C_DIS
LIN {X -0.051,Y -547.808,Z 688.299,A 0.000,B 0.000,C 90.000,E1 269.771} C_DIS
LIN {X 0.182,Y -547.013,Z 688.291,A 0.000,B 0.000,C 90.000,E1 268.339} C_DIS
LIN {X -0.068,Y -546.003,Z 688.282,A 0.000,B 0.000,C 90.000,E1 266.674} C_DIS
LIN {X 0.240,Y -544.581,Z 688.271,A 0.000,B 0.000,C 90.000,E1 264.666} C_DIS
LIN {X -0.030,Y -543.442,Z 688.263,A 0.000,B 0.000,C 90.000,E1 263.280} C_DIS
LIN {X -0.159,Y -541.378,Z 688.252,A 0.000,B 0.000,C 90.000,E1 261.310} C_DIS
LIN {X -0.134,Y -538.758,Z 688.236,A 0.000,B 0.000,C 90.000,E1 258.465} C_DIS
LIN {X -0.080,Y -537.059,Z 688.225,A 0.000,B 0.000,C 90.000,E1 256.464} C_DIS
LIN {X -0.177,Y -535.795,Z 688.217,A 0.000,B 0.000,C 90.000,E1 255.046} C_DIS
LIN {X 0.161,Y -534.657,Z 688.211,A 0.000,B 0.000,C 90.000,E1 253.866} C_DIS
LIN {X -0.166,Y -532.898,Z 688.201,A 0.000,B 0.000,C 90.000,E1 252.181} C_DIS
LIN {X 0.149,Y -531.204,Z 688.191,A 0.000,B 0.000,C 90.000,E1 250.423} C_DIS
LIN {X 0.042,Y -530.214,Z 688.187,A 0.000,B 0.000,C 90.000,E1 249.571} C_DIS
LIN {X -0.021,Y -527.816,Z 688.177,A 0.000,B 0.000,C 90.000,E1 247.847} C_DIS
LIN {X -0.105,Y -525.759,Z 688.169,A 0.000,B 0.000,C 90.000,E1 246.410} C_DIS
LIN {X -0.227,Y -523.348,Z 688.161,A 0.000,B 0.000,C 90.000,E1 244.973} C_DIS
LIN {X -0.008,Y -521.898,Z 688.156,A 0.000,B 0.000,C 90.000,E1 244.076} C_DIS
LIN {X 0.012,Y -519.081,Z 688.148,A 0.000,B 0.000,C 90.000,E1 242.615} C_DIS
LIN {X 0.118,Y -515.633,Z 688.138,A 0.000,B 0.000,C 90.000,E1 240.845} C_DIS
LIN {X 0.147,Y -513.133,Z 688.132,A 0.000,B 0.000,C 90.000,E1 239.665} C_DIS
LIN {X 0.034,Y -509.983,Z 688.123,A 0.000,B 0.000,C 90.000,E1 238.201} C_DIS
LIN {X -0.196,Y -507.410,Z 688.117,A 0.000,B 0.000,C 90.000,E1 237.041} C_DIS
LIN {X 0.133,Y -504.012,Z 688.109,A 0.000,B 0.000,C 90.000,E1 235.515} C_DIS
LIN {X -0.013,Y -500.533,Z 688.100,A 0.000,B 0.000,C 90.000,E1 234.036} C_DIS
LIN {X -0.098,Y -497.599,Z 688.094,A 0.000,B 0.000,C 90.000,E1 232.844} C_DIS
LIN {X 0.092,Y -493.119,Z 688.083,A 0.000,B 0.000,C 90.000,E1 231.009} C_DIS
LIN {X -0.035,Y -489.449,Z 688.075,A 0.000,B 0.000,C 90.000,E1 229.504} C_DIS
LIN {X -0.265,Y -484.448,Z 688.063,A 0.000,B 0.000,C 90.000,E1 227.391} C_DIS
LIN {X 0.008,Y -479.515,Z 688.051,A 0.000,B 0.000,C 90.000,E1 225.202} C_DIS
LIN {X 0.259,Y -475.883,Z 688.043,A 0.000,B 0.000,C 90.000,E1 223.623} C_DIS
LIN {X -0.011,Y -470.942,Z 688.030,A 0.000,B 0.000,C 90.000,E1 221.472} C_DIS
LIN {X 0.120,Y -467.611,Z 688.022,A 0.000,B 0.000,C 90.000,E1 219.886} C_DIS
LIN {X -0.065,Y -463.589,Z 688.011,A 0.000,B 0.000,C 90.000,E1 218.016} C_DIS
LIN {X -0.202,Y -456.789,Z 687.992,A 0.000,B 0.000,C 90.000,E1 214.532} C_DIS
LIN {X 0.091,Y -454.283,Z 687.985,A 0.000,B 0.000,C 90.000,E1 213.214} C_DIS
LIN {X 0.275,Y -450.609,Z 687.974,A 0.000,B 0.000,C 90.000,E1 211.258} C_DIS
LIN {X -0.006,Y -446.345,Z 687.961,A 0.000,B 0.000,C 90.000,E1 209.027} C_DIS
LIN {X -0.053,Y -442.830,Z 687.950,A 0.000,B 0.000,C 90.000,E1 207.078} C_DIS
LIN {X 0.199,Y -439.269,Z 687.940,A 0.000,B 0.000,C 90.000,E1 205.079} C_DIS
LIN {X 0.137,Y -436.847,Z 687.932,A 0.000,B 0.000,C 90.000,E1 203.770} C_DIS
LIN {X -0.128,Y -433.837,Z 687.923,A 0.000,B 0.000,C 90.000,E1 202.153} C_DIS
LIN {X -0.054,Y -430.827,Z 687.914,A 0.000,B 0.000,C 90.000,E1 200.482} C_DIS
LIN {X -0.131,Y -427.131,Z 687.903,A 0.000,B 0.000,C 90.000,E1 198.489} C_DIS
LIN {X -0.105,Y -423.029,Z 687.890,A 0.000,B 0.000,C 90.000,E1 196.134} C_DIS
LIN {X 0.039,Y -420.139,Z 687.880,A 0.000,B 0.000,C 90.000,E1 194.426} C_DIS
LIN {X 0.133,Y -417.106,Z 687.871,A 0.000,B 0.000,C 90.000,E1 192.715} C_DIS
LIN {X 0.201,Y -413.744,Z 687.859,A 0.000,B 0.000,C 90.000,E1 190.658} C_DIS
LIN {X -0.007,Y -411.020,Z 687.850,A 0.000,B 0.000,C 90.000,E1 188.973} C_DIS
LIN {X 0.067,Y -407.351,Z 687.836,A 0.000,B 0.000,C 90.000,E1 186.549} C_DIS
LIN {X -0.003,Y -403.441,Z 687.821,A 0.000,B 0.000,C 90.000,E1 183.784} C_DIS
LIN {X 0.117,Y -400.012,Z 687.806,A 0.000,B 0.000,C 90.000,E1 180.974} C_DIS
LIN {X 0.123,Y -397.199,Z 687.790,A 0.000,B 0.000,C 90.000,E1 178.165} C_DIS
LIN {X 0.055,Y -394.982,Z 687.774,A 0.000,B 0.000,C 90.000,E1 175.355} C_DIS
LIN {X -0.167,Y -392.814,Z 687.751,A 0.000,B 0.000,C 90.000,E1 171.141} C_DIS
LIN {X -0.008,Y -392.177,Z 687.737,A 0.000,B 0.000,C 90.000,E1 168.634} C_DIS
LIN {X -0.111,Y -391.963,Z 687.729,A 0.000,B 0.000,C 90.000,E1 167.229} C_DIS
LIN {X -0.155,Y -391.400,Z 687.713,A 0.000,B 0.000,C 90.000,E1 164.393} C_DIS
LIN {X -0.035,Y -391.319,Z 687.703,A 0.000,B 0.000,C 90.000,E1 162.598} C_DIS
LIN {X -0.120,Y -391.367,Z 687.691,A 0.000,B 0.000,C 90.000,E1 160.477} C_DIS
LIN {X -0.027,Y -391.516,Z 687.678,A 0.000,B 0.000,C 90.000,E1 157.975} C_DIS
LIN {X -0.045,Y -391.714,Z 687.666,A 0.000,B 0.000,C 90.000,E1 155.845} C_DIS
LIN {X 0.133,Y -391.923,Z 687.652,A 0.000,B 0.000,C 90.000,E1 153.332} C_DIS
LIN {X 0.088,Y -392.274,Z 687.642,A 0.000,B 0.000,C 90.000,E1 151.563} C_DIS
LIN {X 0.059,Y -392.738,Z 687.632,A 0.000,B 0.000,C 90.000,E1 149.793} C_DIS
LIN {X 0.092,Y -393.387,Z 687.620,A 0.000,B 0.000,C 90.000,E1 147.661} C_DIS
LIN {X 0.009,Y -394.290,Z 687.609,A 0.000,B 0.000,C 90.000,E1 145.548} C_DIS
LIN {X 0.024,Y -396.084,Z 687.593,A 0.000,B 0.000,C 90.000,E1 142.718} C_DIS
LIN {X -0.145,Y -397.972,Z 687.579,A 0.000,B 0.000,C 90.000,E1 140.275} C_DIS
LIN {X 0.083,Y -399.566,Z 687.569,A 0.000,B 0.000,C 90.000,E1 138.485} C_DIS
LIN {X -0.237,Y -402.262,Z 687.554,A 0.000,B 0.000,C 90.000,E1 135.729} C_DIS
LIN {X -0.194,Y -404.086,Z 687.548,A 0.000,B 0.000,C 90.000,E1 134.676} C_DIS
LIN {X 0.122,Y -405.449,Z 687.545,A 0.000,B 0.000,C 90.000,E1 134.109} C_DIS
LIN {X 0.136,Y -407.868,Z 687.542,A 0.000,B 0.000,C 90.000,E1 133.542} C_DIS
LIN {X 0.166,Y -411.383,Z 687.539,A 0.000,B 0.000,C 90.000,E1 133.014} C_DIS
LIN {X 0.183,Y -415.903,Z 687.536,A 0.000,B 0.000,C 90.000,E1 132.528} C_DIS
LIN {X 0.013,Y -433.748,Z 687.528,A 0.000,B 0.000,C 90.000,E1 130.943} C_DIS
LIN {X -0.221,Y -450.855,Z 687.520,A 0.000,B 0.000,C 90.000,E1 129.564} C_DIS
LIN {X 0.071,Y -463.169,Z 687.514,A 0.000,B 0.000,C 90.000,E1 128.543} C_DIS
LIN {X 0.000,Y -469.091,Z 687.511,A 0.000,B 0.000,C 90.000,E1 128.051} C_DIS
LIN {X 0.062,Y -477.910,Z 687.507,A 0.000,B 0.000,C 90.000,E1 127.282} C_DIS
LIN {X -0.001,Y -486.416,Z 687.503,A 0.000,B 0.000,C 90.000,E1 126.503} C_DIS
LIN {X 0.085,Y -492.078,Z 687.500,A 0.000,B 0.000,C 90.000,E1 125.964} C_DIS
LIN {X 0.021,Y -501.553,Z 687.495,A 0.000,B 0.000,C 90.000,E1 125.025} C_DIS
LIN {X 0.045,Y -506.680,Z 687.492,A 0.000,B 0.000,C 90.000,E1 124.485} C_DIS
LIN {X 0.083,Y -511.851,Z 687.489,A 0.000,B 0.000,C 90.000,E1 123.913} C_DIS
LIN {X -0.169,Y -515.713,Z 687.486,A 0.000,B 0.000,C 90.000,E1 123.499} C_DIS
LIN {X 0.121,Y -521.575,Z 687.482,A 0.000,B 0.000,C 90.000,E1 122.752} C_DIS
LIN {X 0.280,Y -524.728,Z 687.480,A 0.000,B 0.000,C 90.000,E1 122.339} C_DIS
LIN {X -0.252,Y -529.830,Z 687.476,A 0.000,B 0.000,C 90.000,E1 121.671} C_DIS
LIN {X 0.142,Y -533.652,Z 687.473,A 0.000,B 0.000,C 90.000,E1 121.052} C_DIS
LIN {X 0.292,Y -537.130,Z 687.469,A 0.000,B 0.000,C 90.000,E1 120.463} C_DIS
LIN {X -0.272,Y -541.645,Z 687.465,A 0.000,B 0.000,C 90.000,E1 119.667} C_DIS
LIN {X -0.190,Y -545.149,Z 687.461,A 0.000,B 0.000,C 90.000,E1 118.949} C_DIS
LIN {X -0.075,Y -548.397,Z 687.457,A 0.000,B 0.000,C 90.000,E1 118.231} C_DIS
LIN {X 0.187,Y -550.883,Z 687.454,A 0.000,B 0.000,C 90.000,E1 117.641} C_DIS
LIN {X -0.015,Y -554.304,Z 687.449,A 0.000,B 0.000,C 90.000,E1 116.821} C_DIS
LIN {X -0.146,Y -558.474,Z 687.443,A 0.000,B 0.000,C 90.000,E1 115.720} C_DIS
LIN {X -0.267,Y -561.411,Z 687.438,A 0.000,B 0.000,C 90.000,E1 114.899} C_DIS
LIN {X 0.158,Y -564.072,Z 687.434,A 0.000,B 0.000,C 90.000,E1 114.027} C_DIS
LIN {X 0.099,Y -566.489,Z 687.429,A 0.000,B 0.000,C 90.000,E1 113.206} C_DIS
LIN {X 0.058,Y -568.579,Z 687.424,A 0.000,B 0.000,C 90.000,E1 112.386} C_DIS
LIN {X 0.169,Y -570.929,Z 687.418,A 0.000,B 0.000,C 90.000,E1 111.280} C_DIS
LIN {X 0.116,Y -573.113,Z 687.412,A 0.000,B 0.000,C 90.000,E1 110.194} C_DIS
LIN {X -0.250,Y -576.027,Z 687.403,A 0.000,B 0.000,C 90.000,E1 108.598} C_DIS
LIN {X -0.030,Y -578.483,Z 687.396,A 0.000,B 0.000,C 90.000,E1 107.221} C_DIS
LIN {X 0.238,Y -580.886,Z 687.388,A 0.000,B 0.000,C 90.000,E1 105.843} C_DIS
LIN {X -0.174,Y -583.120,Z 687.381,A 0.000,B 0.000,C 90.000,E1 104.537} C_DIS
LIN {X 0.013,Y -585.306,Z 687.373,A 0.000,B 0.000,C 90.000,E1 103.175} C_DIS
LIN {X -0.149,Y -587.098,Z 687.367,A 0.000,B 0.000,C 90.000,E1 102.119} C_DIS
LIN {X 0.117,Y -589.750,Z 687.358,A 0.000,B 0.000,C 90.000,E1 100.489} C_DIS
LIN {X -0.089,Y -591.432,Z 687.352,A 0.000,B 0.000,C 90.000,E1 99.443} C_DIS
LIN {X -0.275,Y -593.030,Z 687.347,A 0.000,B 0.000,C 90.000,E1 98.398} C_DIS
LIN {X 0.027,Y -595.252,Z 687.338,A 0.000,B 0.000,C 90.000,E1 96.777} C_DIS
LIN {X 0.299,Y -597.287,Z 687.329,A 0.000,B 0.000,C 90.000,E1 95.163} C_DIS
LIN {X -0.268,Y -598.930,Z 687.322,A 0.000,B 0.000,C 90.000,E1 93.898} C_DIS
LIN {X 0.108,Y -600.041,Z 687.316,A 0.000,B 0.000,C 90.000,E1 92.808} C_DIS
LIN {X 0.144,Y -601.243,Z 687.308,A 0.000,B 0.000,C 90.000,E1 91.489} C_DIS
LIN {X -0.065,Y -602.040,Z 687.303,A 0.000,B 0.000,C 90.000,E1 90.458} C_DIS
LIN {X -0.261,Y -602.676,Z 687.297,A 0.000,B 0.000,C 90.000,E1 89.427} C_DIS
LIN {X 0.076,Y -603.275,Z 687.288,A 0.000,B 0.000,C 90.000,E1 87.822} C_DIS
LIN {X 0.234,Y -603.481,Z 687.284,A 0.000,B 0.000,C 90.000,E1 87.020} C_DIS
LIN {X 0.010,Y -603.700,Z 687.275,A 0.000,B 0.000,C 90.000,E1 85.469} C_DIS
LIN {X 0.145,Y -603.640,Z 687.268,A 0.000,B 0.000,C 90.000,E1 84.147} C_DIS
LIN {X 0.034,Y -603.420,Z 687.262,A 0.000,B 0.000,C 90.000,E1 83.109} C_DIS
LIN {X 0.227,Y -602.995,Z 687.255,A 0.000,B 0.000,C 90.000,E1 81.781} C_DIS
LIN {X -0.122,Y -602.633,Z 687.250,A 0.000,B 0.000,C 90.000,E1 81.027} C_DIS
LIN {X -0.164,Y -601.861,Z 687.244,A 0.000,B 0.000,C 90.000,E1 79.982} C_DIS
LIN {X -0.105,Y -601.000,Z 687.238,A 0.000,B 0.000,C 90.000,E1 78.926} C_DIS
LIN {X -0.156,Y -599.412,Z 687.230,A 0.000,B 0.000,C 90.000,E1 77.353} C_DIS
LIN {X 0.011,Y -598.293,Z 687.224,A 0.000,B 0.000,C 90.000,E1 76.284} C_DIS
LIN {X 0.018,Y -596.419,Z 687.215,A 0.000,B 0.000,C 90.000,E1 74.700} C_DIS
LIN {X 0.145,Y -595.061,Z 687.209,A 0.000,B 0.000,C 90.000,E1 73.630} C_DIS
LIN {X 0.119,Y -593.213,Z 687.202,A 0.000,B 0.000,C 90.000,E1 72.308} C_DIS
LIN {X -0.184,Y -591.660,Z 687.196,A 0.000,B 0.000,C 90.000,E1 71.275} C_DIS
LIN {X -0.069,Y -589.459,Z 687.189,A 0.000,B 0.000,C 90.000,E1 69.934} C_DIS
LIN {X 0.005,Y -586.978,Z 687.181,A 0.000,B 0.000,C 90.000,E1 68.592} C_DIS
LIN {X -0.168,Y -584.741,Z 687.175,A 0.000,B 0.000,C 90.000,E1 67.539} C_DIS
LIN {X 0.162,Y -582.193,Z 687.169,A 0.000,B 0.000,C 90.000,E1 66.433} C_DIS
LIN {X 0.151,Y -579.341,Z 687.163,A 0.000,B 0.000,C 90.000,E1 65.357} C_DIS
LIN {X 0.250,Y -577.024,Z 687.159,A 0.000,B 0.000,C 90.000,E1 64.537} C_DIS
LIN {X -0.193,Y -574.496,Z 687.154,A 0.000,B 0.000,C 90.000,E1 63.768} C_DIS
LIN {X -0.050,Y -570.874,Z 687.148,A 0.000,B 0.000,C 90.000,E1 62.666} C_DIS
LIN {X -0.049,Y -567.902,Z 687.144,A 0.000,B 0.000,C 90.000,E1 61.847} C_DIS
LIN {X 0.180,Y -564.767,Z 687.139,A 0.000,B 0.000,C 90.000,E1 61.001} C_DIS
LIN {X -0.116,Y -561.231,Z 687.134,A 0.000,B 0.000,C 90.000,E1 60.205} C_DIS
LIN {X 0.139,Y -558.080,Z 687.131,A 0.000,B 0.000,C 90.000,E1 59.488} C_DIS
LIN {X 0.169,Y -554.411,Z 687.127,A 0.000,B 0.000,C 90.000,E1 58.791} C_DIS
LIN {X -0.117,Y -550.306,Z 687.123,A 0.000,B 0.000,C 90.000,E1 58.122} C_DIS
LIN {X 0.024,Y -545.795,Z 687.119,A 0.000,B 0.000,C 90.000,E1 57.406} C_DIS
LIN {X -0.073,Y -542.928,Z 687.117,A 0.000,B 0.000,C 90.000,E1 56.993} C_DIS
LIN {X -0.024,Y -538.644,Z 687.113,A 0.000,B 0.000,C 90.000,E1 56.421} C_DIS
LIN {X -0.161,Y -534.053,Z 687.110,A 0.000,B 0.000,C 90.000,E1 55.881} C_DIS
LIN {X -0.047,Y -529.129,Z 687.107,A 0.000,B 0.000,C 90.000,E1 55.341} C_DIS
LIN {X 0.046,Y -523.590,Z 687.105,A 0.000,B 0.000,C 90.000,E1 54.815} C_DIS
LIN {X 0.061,Y -519.216,Z 687.102,A 0.000,B 0.000,C 90.000,E1 54.436} C_DIS
LIN {X -0.184,Y -513.004,Z 687.100,A 0.000,B 0.000,C 90.000,E1 53.989} C_DIS
LIN {X 0.040,Y -508.139,Z 687.098,A 0.000,B 0.000,C 90.000,E1 53.623} C_DIS
LIN {X -0.200,Y -499.892,Z 687.095,A 0.000,B 0.000,C 90.000,E1 53.130} C_DIS
LIN {X -0.185,Y -491.575,Z 687.092,A 0.000,B 0.000,C 90.000,E1 52.637} C_DIS
LIN {X -0.147,Y -474.967,Z 687.087,A 0.000,B 0.000,C 90.000,E1 51.698} C_DIS
LIN {X -0.104,Y -456.832,Z 687.081,A 0.000,B 0.000,C 90.000,E1 50.642} C_DIS
LIN {X -0.132,Y -437.409,Z 687.075,A 0.000,B 0.000,C 90.000,E1 49.461} C_DIS
LIN {X -0.005,Y -427.900,Z 687.071,A 0.000,B 0.000,C 90.000,E1 48.809} C_DIS
LIN {X 0.029,Y -426.350,Z 687.071,A 0.000,B 0.000,C 90.000,E1 48.690} C_DIS
LIN {X 0.005,Y -426.330,Z 687.071,A 0.000,B 0.000,C 90.000,E1 48.690} C_DIS
LIN {X -0.186,Y -418.768,Z 687.049,A 0.000,B 0.000,C 90.000,E1 44.919} C_DIS
LIN {X 0.096,Y -412.978,Z 687.035,A 0.000,B 0.000,C 90.000,E1 42.324} C_DIS
LIN {X 0.115,Y -413.003,Z 687.023,A 0.000,B 0.000,C 90.000,E1 40.092} C_DIS
LIN {X 0.108,Y -413.793,Z 687.004,A 0.000,B 0.000,C 90.000,E1 36.664} C_DIS
LIN {X -0.086,Y -414.581,Z 686.994,A 0.000,B 0.000,C 90.000,E1 34.978} C_DIS
LIN {X 0.137,Y -415.234,Z 686.987,A 0.000,B 0.000,C 90.000,E1 33.579} C_DIS
LIN {X 0.030,Y -416.339,Z 686.975,A 0.000,B 0.000,C 90.000,E1 31.544} C_DIS
LIN {X -0.221,Y -417.247,Z 686.966,A 0.000,B 0.000,C 90.000,E1 29.873} C_DIS
LIN {X -0.022,Y -418.646,Z 686.953,A 0.000,B 0.000,C 90.000,E1 27.462} C_DIS
LIN {X 0.017,Y -420.300,Z 686.939,A 0.000,B 0.000,C 90.000,E1 25.079} C_DIS
LIN {X 0.069,Y -422.817,Z 686.922,A 0.000,B 0.000,C 90.000,E1 22.025} C_DIS
LIN {X -0.060,Y -424.473,Z 686.913,A 0.000,B 0.000,C 90.000,E1 20.355} C_DIS
LIN {X -0.050,Y -426.037,Z 686.904,A 0.000,B 0.000,C 90.000,E1 18.671} C_DIS
LIN {X -0.004,Y -428.223,Z 686.891,A 0.000,B 0.000,C 90.000,E1 16.315} C_DIS
LIN {X 0.056,Y -430.298,Z 686.880,A 0.000,B 0.000,C 90.000,E1 14.300} C_DIS
LIN {X 0.064,Y -432.518,Z 686.868,A 0.000,B 0.000,C 90.000,E1 12.299} C_DIS
LIN {X 0.160,Y -435.216,Z 686.856,A 0.000,B 0.000,C 90.000,E1 9.962} C_DIS
LIN {X -0.110,Y -438.465,Z 686.841,A 0.000,B 0.000,C 90.000,E1 7.352} C_DIS
LIN {X -0.071,Y -440.229,Z 686.833,A 0.000,B 0.000,C 90.000,E1 6.030} C_DIS
LIN {X -0.184,Y -444.387,Z 686.817,A 0.000,B 0.000,C 90.000,E1 3.094} C_DIS
LIN {X 0.046,Y -448.528,Z 686.803,A 0.000,B 0.000,C 90.000,E1 0.458} C_DIS
LIN {X -0.210,Y -453.062,Z 686.788,A 0.000,B 0.000,C 90.000,E1 357.879} C_DIS
LIN {X 0.042,Y -455.552,Z 686.781,A 0.000,B 0.000,C 90.000,E1 356.560} C_DIS
LIN {X 0.088,Y -458.635,Z 686.772,A 0.000,B 0.000,C 90.000,E1 354.951} C_DIS
LIN {X -0.035,Y -462.324,Z 686.761,A 0.000,B 0.000,C 90.000,E1 353.053} C_DIS
LIN {X -0.223,Y -465.355,Z 686.753,A 0.000,B 0.000,C 90.000,E1 351.489} C_DIS
LIN {X 0.189,Y -468.330,Z 686.744,A 0.000,B 0.000,C 90.000,E1 349.859} C_DIS
LIN {X -0.083,Y -470.568,Z 686.737,A 0.000,B 0.000,C 90.000,E1 348.634} C_DIS
LIN {X -0.103,Y -473.915,Z 686.726,A 0.000,B 0.000,C 90.000,E1 346.756} C_DIS
LIN {X 0.064,Y -477.367,Z 686.716,A 0.000,B 0.000,C 90.000,E1 344.866} C_DIS
LIN {X -0.028,Y -480.909,Z 686.706,A 0.000,B 0.000,C 90.000,E1 343.015} C_DIS
LIN {X -0.048,Y -485.242,Z 686.694,A 0.000,B 0.000,C 90.000,E1 340.859} C_DIS
LIN {X -0.149,Y -488.341,Z 686.685,A 0.000,B 0.000,C 90.000,E1 339.337} C_DIS
LIN {X -0.018,Y -491.439,Z 686.677,A 0.000,B 0.000,C 90.000,E1 337.794} C_DIS
LIN {X -0.084,Y -494.556,Z 686.668,A 0.000,B 0.000,C 90.000,E1 336.282} C_DIS
LIN {X 0.056,Y -496.417,Z 686.663,A 0.000,B 0.000,C 90.000,E1 335.357} C_DIS
LIN {X -0.295,Y -497.984,Z 686.660,A 0.000,B 0.000,C 90.000,E1 334.793} C_DIS
LIN {X 0.226,Y -499.501,Z 686.657,A 0.000,B 0.000,C 90.000,E1 334.280} C_DIS
LIN {X -0.167,Y -500.985,Z 686.656,A 0.000,B 0.000,C 90.000,E1 334.024} C_DIS
LIN {X -0.074,Y -503.939,Z 686.653,A 0.000,B 0.000,C 90.000,E1 333.563} C_DIS
LIN {X 0.054,Y -505.673,Z 686.652,A 0.000,B 0.000,C 90.000,E1 333.332} C_DIS
LIN {X -0.045,Y -510.827,Z 686.649,A 0.000,B 0.000,C 90.000,E1 332.871} C_DIS
LIN {X 0.148,Y -519.242,Z 686.646,A 0.000,B 0.000,C 90.000,E1 332.231} C_DIS
LIN {X -0.109,Y -531.623,Z 686.641,A 0.000,B 0.000,C 90.000,E1 331.435} C_DIS
LIN {X -0.053,Y -537.699,Z 686.639,A 0.000,B 0.000,C 90.000,E1 331.001} C_DIS
LIN {X 0.158,Y -543.596,Z 686.636,A 0.000,B 0.000,C 90.000,E1 330.539} C_DIS
LIN {X 0.100,Y -549.329,Z 686.634,A 0.000,B 0.000,C 90.000,E1 330.078} C_DIS
LIN {X 0.242,Y -557.699,Z 686.630,A 0.000,B 0.000,C 90.000,E1 329.331} C_DIS
LIN {X -0.069,Y -564.187,Z 686.626,A 0.000,B 0.000,C 90.000,E1 328.742} C_DIS
LIN {X -0.315,Y -571.971,Z 686.622,A 0.000,B 0.000,C 90.000,E1 327.995} C_DIS
LIN {X 0.000,Y -578.121,Z 686.619,A 0.000,B 0.000,C 90.000,E1 327.327} C_DIS
LIN {X -0.262,Y -586.808,Z 686.613,A 0.000,B 0.000,C 90.000,E1 326.421} C_DIS
LIN {X 0.010,Y -595.358,Z 686.608,A 0.000,B 0.000,C 90.000,E1 325.468} C_DIS
LIN {X -0.045,Y -601.288,Z 686.605,A 0.000,B 0.000,C 90.000,E1 324.815} C_DIS
LIN {X 0.103,Y -605.670,Z 686.602,A 0.000,B 0.000,C 90.000,E1 324.276} C_DIS
LIN {X -0.214,Y -609.837,Z 686.599,A 0.000,B 0.000,C 90.000,E1 323.783} C_DIS
LIN {X -0.064,Y -615.781,Z 686.594,A 0.000,B 0.000,C 90.000,E1 323.004} C_DIS
LIN {X 0.023,Y -620.442,Z 686.591,A 0.000,B 0.000,C 90.000,E1 322.351} C_DIS
LIN {X -0.025,Y -627.406,Z 686.585,A 0.000,B 0.000,C 90.000,E1 321.331} C_DIS
LIN {X -0.327,Y -631.485,Z 686.582,A 0.000,B 0.000,C 90.000,E1 320.723} C_DIS
LIN {X -0.105,Y -635.355,Z 686.578,A 0.000,B 0.000,C 90.000,E1 320.070} C_DIS
LIN {X -0.046,Y -642.065,Z 686.572,A 0.000,B 0.000,C 90.000,E1 318.933} C_DIS
LIN {X 0.122,Y -647.650,Z 686.566,A 0.000,B 0.000,C 90.000,E1 317.919} C_DIS
LIN {X -0.021,Y -651.712,Z 686.562,A 0.000,B 0.000,C 90.000,E1 317.187} C_DIS
LIN {X 0.279,Y -656.163,Z 686.557,A 0.000,B 0.000,C 90.000,E1 316.296} C_DIS
LIN {X 0.184,Y -659.656,Z 686.553,A 0.000,B 0.000,C 90.000,E1 315.567} C_DIS
LIN {X 0.107,Y -664.030,Z 686.548,A 0.000,B 0.000,C 90.000,E1 314.595} C_DIS
LIN {X 0.083,Y -669.138,Z 686.541,A 0.000,B 0.000,C 90.000,E1 313.380} C_DIS
LIN {X 0.193,Y -675.181,Z 686.533,A 0.000,B 0.000,C 90.000,E1 311.919} C_DIS
LIN {X -0.126,Y -679.803,Z 686.526,A 0.000,B 0.000,C 90.000,E1 310.744} C_DIS
LIN {X 0.089,Y -683.027,Z 686.521,A 0.000,B 0.000,C 90.000,E1 309.769} C_DIS
LIN {X -0.084,Y -686.009,Z 686.516,A 0.000,B 0.000,C 90.000,E1 308.830} C_DIS
LIN {X -0.214,Y -688.600,Z 686.510,A 0.000,B 0.000,C 90.000,E1 307.890} C_DIS
LIN {X -0.309,Y -690.980,Z 686.505,A 0.000,B 0.000,C 90.000,E1 306.950} C_DIS
LIN {X 0.182,Y -693.070,Z 686.500,A 0.000,B 0.000,C 90.000,E1 305.964} C_DIS
LIN {X 0.089,Y -694.452,Z 686.496,A 0.000,B 0.000,C 90.000,E1 305.264} C_DIS
LIN {X 0.009,Y -695.729,Z 686.492,A 0.000,B 0.000,C 90.000,E1 304.565} C_DIS
LIN {X -0.060,Y -696.880,Z 686.488,A 0.000,B 0.000,C 90.000,E1 303.865} C_DIS
LIN {X -0.124,Y -697.874,Z 686.484,A 0.000,B 0.000,C 90.000,E1 303.166} C_DIS
LIN {X 0.065,Y -699.050,Z 686.479,A 0.000,B 0.000,C 90.000,E1 302.212} C_DIS
LIN {X -0.072,Y -700.372,Z 686.473,A 0.000,B 0.000,C 90.000,E1 301.052} C_DIS
LIN {X 0.118,Y -700.986,Z 686.469,A 0.000,B 0.000,C 90.000,E1 300.335} C_DIS
LIN {X 0.257,Y -701.759,Z 686.462,A 0.000,B 0.000,C 90.000,E1 299.155} C_DIS
LIN {X 0.345,Y -702.644,Z 686.453,A 0.000,B 0.000,C 90.000,E1 297.513} C_DIS
LIN {X 0.090,Y -703.919,Z 686.443,A 0.000,B 0.000,C 90.000,E1 295.668} C_DIS
LIN {X 0.024,Y -703.718,Z 686.440,A 0.000,B 0.000,C 90.000,E1 295.207} C_DIS
LIN {X 0.010,Y -703.500,Z 686.439,A 0.000,B 0.000,C 90.000,E1 294.975} C_DIS
LIN {X -0.064,Y -702.114,Z 686.436,A 0.000,B 0.000,C 90.000,E1 294.515} C_DIS
LIN {X 0.215,Y -701.131,Z 686.435,A 0.000,B 0.000,C 90.000,E1 294.259} C_DIS
LIN {X 0.066,Y -700.231,Z 686.434,A 0.000,B 0.000,C 90.000,E1 294.155} C_DIS
LIN {X -0.301,Y -698.091,Z 686.433,A 0.000,B 0.000,C 90.000,E1 293.951} C_DIS
LIN {X -0.018,Y -695.667,Z 686.432,A 0.000,B 0.000,C 90.000,E1 293.695} C_DIS
LIN {X 0.128,Y -694.007,Z 686.431,A 0.000,B 0.000,C 90.000,E1 293.567} C_DIS
LIN {X -0.065,Y -689.271,Z 686.430,A 0.000,B 0.000,C 90.000,E1 293.387} C_DIS
LIN {X -0.220,Y -687.258,Z 686.430,A 0.000,B 0.000,C 90.000,E1 293.334} C_DIS
LIN {X 0.201,Y -681.013,Z 686.429,A 0.000,B 0.000,C 90.000,E1 293.153} C_DIS
LIN {X -0.002,Y -678.996,Z 686.429,A 0.000,B 0.000,C 90.000,E1 293.131} C_DIS
LIN {X 0.190,Y -661.267,Z 686.427,A 0.000,B 0.000,C 90.000,E1 292.898} C_DIS
LIN {X 0.082,Y -647.564,Z 686.426,A 0.000,B 0.000,C 90.000,E1 292.695} C_DIS
LIN {X -0.187,Y -634.239,Z 686.425,A 0.000,B 0.000,C 90.000,E1 292.461} C_DIS
LIN {X 0.155,Y -617.681,Z 686.422,A 0.000,B 0.000,C 90.000,E1 292.025} C_DIS
LIN {X -0.116,Y -593.683,Z 686.419,A 0.000,B 0.000,C 90.000,E1 291.354} C_DIS
LIN {X 0.118,Y -576.272,Z 686.416,A 0.000,B 0.000,C 90.000,E1 290.791} C_DIS
LIN {X 0.132,Y -562.268,Z 686.413,A 0.000,B 0.000,C 90.000,E1 290.375} C_DIS
LIN {X -0.058,Y -557.455,Z 686.412,A 0.000,B 0.000,C 90.000,E1 290.174} C_DIS
LIN {X 0.013,Y -555.566,Z 686.411,A 0.000,B 0.000,C 90.000,E1 289.993} C_DIS
LIN {X -0.027,Y -555.531,Z 686.411,A 0.000,B 0.000,C 90.000,E1 289.993} C_DIS
LIN {X -0.033,Y -554.874,Z 686.410,A 0.000,B 0.000,C 90.000,E1 289.758} C_DIS
LIN {X 0.254,Y -554.473,Z 686.408,A 0.000,B 0.000,C 90.000,E1 289.450} C_DIS
LIN {X 0.115,Y -554.165,Z 686.405,A 0.000,B 0.000,C 90.000,E1 288.906} C_DIS
LIN {X 0.107,Y -553.762,Z 686.397,A 0.000,B 0.000,C 90.000,E1 287.511} C_DIS
LIN {X 0.149,Y -553.144,Z 686.387,A 0.000,B 0.000,C 90.000,E1 285.552} C_DIS
LIN {X 0.063,Y -552.482,Z 686.377,A 0.000,B 0.000,C 90.000,E1 283.883} C_DIS
LIN {X 0.118,Y -551.840,Z 686.369,A 0.000,B 0.000,C 90.000,E1 282.479} C_DIS
LIN {X 0.051,Y -551.277,Z 686.363,A 0.000,B 0.000,C 90.000,E1 281.366} C_DIS
LIN {X 0.085,Y -550.619,Z 686.355,A 0.000,B 0.000,C 90.000,E1 279.962} C_DIS
LIN {X 0.245,Y -549.793,Z 686.343,A 0.000,B 0.000,C 90.000,E1 277.701} C_DIS
LIN {X 0.112,Y -549.384,Z 686.334,A 0.000,B 0.000,C 90.000,E1 276.030} C_DIS
LIN {X -0.026,Y -549.178,Z 686.324,A 0.000,B 0.000,C 90.000,E1 274.359} C_DIS
LIN {X 0.202,Y -549.110,Z 686.318,A 0.000,B 0.000,C 90.000,E1 273.212} C_DIS
LIN {X -0.119,Y -548.868,Z 686.312,A 0.000,B 0.000,C 90.000,E1 272.121} C_DIS
LIN {X 0.051,Y -548.634,Z 686.307,A 0.000,B 0.000,C 90.000,E1 271.260} C_DIS
LIN {X 0.252,Y -548.064,Z 686.301,A 0.000,B 0.000,C 90.000,E1 270.115} C_DIS
LIN {X -0.011,Y -547.104,Z 686.291,A 0.000,B 0.000,C 90.000,E1 268.453} C_DIS
LIN {X -0.257,Y -546.095,Z 686.282,A 0.000,B 0.000,C 90.000,E1 266.788} C_DIS
LIN {X 0.029,Y -544.853,Z 686.273,A 0.000,B 0.000,C 90.000,E1 265.065} C_DIS
LIN {X 0.254,Y -543.774,Z 686.265,A 0.000,B 0.000,C 90.000,E1 263.628} C_DIS
LIN {X -0.194,Y -543.270,Z 686.262,A 0.000,B 0.000,C 90.000,E1 263.109} C_DIS
LIN {X 0.126,Y -541.476,Z 686.252,A 0.000,B 0.000,C 90.000,E1 261.376} C_DIS
LIN {X 0.169,Y -539.073,Z 686.238,A 0.000,B 0.000,C 90.000,E1 258.814} C_DIS
LIN {X -0.017,Y -537.851,Z 686.230,A 0.000,B 0.000,C 90.000,E1 257.409} C_DIS
LIN {X -0.044,Y -536.430,Z 686.221,A 0.000,B 0.000,C 90.000,E1 255.700} C_DIS
LIN {X -0.208,Y -535.392,Z 686.214,A 0.000,B 0.000,C 90.000,E1 254.574} C_DIS
LIN {X 0.031,Y -533.336,Z 686.203,A 0.000,B 0.000,C 90.000,E1 252.543} C_DIS
LIN {X -0.131,Y -531.323,Z 686.192,A 0.000,B 0.000,C 90.000,E1 250.550} C_DIS
LIN {X -0.239,Y -530.352,Z 686.187,A 0.000,B 0.000,C 90.000,E1 249.699} C_DIS
LIN {X -0.174,Y -528.805,Z 686.181,A 0.000,B 0.000,C 90.000,E1 248.539} C_DIS
LIN {X 0.237,Y -526.753,Z 686.173,A 0.000,B 0.000,C 90.000,E1 247.050} C_DIS
LIN {X -0.209,Y -525.491,Z 686.168,A 0.000,B 0.000,C 90.000,E1 246.230} C_DIS
LIN {X 0.039,Y -522.558,Z 686.158,A 0.000,B 0.000,C 90.000,E1 244.460} C_DIS
LIN {X 0.020,Y -520.978,Z 686.153,A 0.000,B 0.000,C 90.000,E1 243.589} C_DIS
LIN {X -0.209,Y -518.125,Z 686.145,A 0.000,B 0.000,C 90.000,E1 242.153} C_DIS
LIN {X -0.030,Y -515.259,Z 686.137,A 0.000,B 0.000,C 90.000,E1 240.667} C_DIS
LIN {X -0.116,Y -510.839,Z 686.126,A 0.000,B 0.000,C 90.000,E1 238.614} C_DIS
LIN {X 0.092,Y -508.276,Z 686.119,A 0.000,B 0.000,C 90.000,E1 237.406} C_DIS
LIN {X 0.320,Y -504.221,Z 686.109,A 0.000,B 0.000,C 90.000,E1 235.595} C_DIS
LIN {X 0.173,Y -500.734,Z 686.101,A 0.000,B 0.000,C 90.000,E1 234.116} C_DIS
LIN {X 0.087,Y -497.780,Z 686.094,A 0.000,B 0.000,C 90.000,E1 232.924} C_DIS
LIN {X 0.277,Y -493.335,Z 686.084,A 0.000,B 0.000,C 90.000,E1 231.090} C_DIS
LIN {X -0.167,Y -489.653,Z 686.076,A 0.000,B 0.000,C 90.000,E1 229.622} C_DIS
LIN {X -0.077,Y -484.640,Z 686.064,A 0.000,B 0.000,C 90.000,E1 227.472} C_DIS
LIN {X -0.142,Y -479.659,Z 686.052,A 0.000,B 0.000,C 90.000,E1 225.324} C_DIS
LIN {X -0.003,Y -476.781,Z 686.045,A 0.000,B 0.000,C 90.000,E1 224.069} C_DIS
LIN {X -0.169,Y -471.086,Z 686.031,A 0.000,B 0.000,C 90.000,E1 221.595} C_DIS
LIN {X -0.041,Y -467.752,Z 686.022,A 0.000,B 0.000,C 90.000,E1 220.011} C_DIS
LIN {X 0.136,Y -463.717,Z 686.012,A 0.000,B 0.000,C 90.000,E1 218.096} C_DIS
LIN {X 0.008,Y -456.911,Z 685.992,A 0.000,B 0.000,C 90.000,E1 214.612} C_DIS
LIN {X 0.304,Y -454.453,Z 685.985,A 0.000,B 0.000,C 90.000,E1 213.293} C_DIS
LIN {X 0.110,Y -450.752,Z 685.974,A 0.000,B 0.000,C 90.000,E1 211.386} C_DIS
LIN {X -0.168,Y -446.469,Z 685.962,A 0.000,B 0.000,C 90.000,E1 209.155} C_DIS
LIN {X -0.063,Y -443.549,Z 685.953,A 0.000,B 0.000,C 90.000,E1 207.513} C_DIS
LIN {X 0.167,Y -440.580,Z 685.944,A 0.000,B 0.000,C 90.000,E1 205.848} C_DIS
LIN {X 0.147,Y -437.646,Z 685.935,A 0.000,B 0.000,C 90.000,E1 204.207} C_DIS
LIN {X -0.104,Y -434.588,Z 685.925,A 0.000,B 0.000,C 90.000,E1 202.589} C_DIS
LIN {X -0.011,Y -431.577,Z 685.916,A 0.000,B 0.000,C 90.000,E1 200.918} C_DIS
LIN {X 0.073,Y -427.897,Z 685.905,A 0.000,B 0.000,C 90.000,E1 198.906} C_DIS
LIN {X -0.072,Y -424.333,Z 685.894,A 0.000,B 0.000,C 90.000,E1 196.913} C_DIS
LIN {X 0.028,Y -422.053,Z 685.886,A 0.000,B 0.000,C 90.000,E1 195.552} C_DIS
LIN {X 0.099,Y -419.731,Z 685.879,A 0.000,B 0.000,C 90.000,E1 194.189} C_DIS
LIN {X 0.071,Y -414.482,Z 685.862,A 0.000,B 0.000,C 90.000,E1 191.130} C_DIS
LIN {X -0.116,Y -411.767,Z 685.852,A 0.000,B 0.000,C 90.000,E1 189.443} C_DIS
LIN {X 0.047,Y -409.045,Z 685.843,A 0.000,B 0.000,C 90.000,E1 187.701} C_DIS
LIN {X 0.089,Y -406.528,Z 685.833,A 0.000,B 0.000,C 90.000,E1 185.967} C_DIS
LIN {X -0.077,Y -402.731,Z 685.818,A 0.000,B 0.000,C 90.000,E1 183.212} C_DIS
LIN {X 0.028,Y -399.418,Z 685.802,A 0.000,B 0.000,C 90.000,E1 180.401} C_DIS
LIN {X 0.175,Y -397.704,Z 685.793,A 0.000,B 0.000,C 90.000,E1 178.625} C_DIS
LIN {X 0.071,Y -395.156,Z 685.775,A 0.000,B 0.000,C 90.000,E1 175.469} C_DIS
LIN {X -0.097,Y -393.117,Z 685.753,A 0.000,B 0.000,C 90.000,E1 171.602} C_DIS
LIN {X -0.055,Y -392.249,Z 685.734,A 0.000,B 0.000,C 90.000,E1 168.049} C_DIS
LIN {X -0.160,Y -391.964,Z 685.726,A 0.000,B 0.000,C 90.000,E1 166.645} C_DIS
LIN {X -0.058,Y -391.584,Z 685.708,A 0.000,B 0.000,C 90.000,E1 163.433} C_DIS
LIN {X -0.162,Y -391.581,Z 685.692,A 0.000,B 0.000,C 90.000,E1 160.604} C_DIS
LIN {X -0.066,Y -391.715,Z 685.678,A 0.000,B 0.000,C 90.000,E1 158.103} C_DIS
LIN {X -0.046,Y -391.961,Z 685.665,A 0.000,B 0.000,C 90.000,E1 155.613} C_DIS
LIN {X 0.102,Y -392.155,Z 685.653,A 0.000,B 0.000,C 90.000,E1 153.461} C_DIS
LIN {X 0.062,Y -392.522,Z 685.643,A 0.000,B 0.000,C 90.000,E1 151.691} C_DIS
LIN {X -0.102,Y -393.027,Z 685.631,A 0.000,B 0.000,C 90.000,E1 149.587} C_DIS
LIN {X -0.059,Y -393.704,Z 685.619,A 0.000,B 0.000,C 90.000,E1 147.454} C_DIS
LIN {X 0.007,Y -394.491,Z 685.609,A 0.000,B 0.000,C 90.000,E1 145.674} C_DIS
LIN {X 0.130,Y -396.404,Z 685.592,A 0.000,B 0.000,C 90.000,E1 142.477} C_DIS
LIN {X -0.020,Y -398.284,Z 685.578,A 0.000,B 0.000,C 90.000,E1 140.033} C_DIS
LIN {X 0.217,Y -399.835,Z 685.568,A 0.000,B 0.000,C 90.000,E1 138.243} C_DIS
LIN {X 0.087,Y -402.108,Z 685.555,A 0.000,B 0.000,C 90.000,E1 135.810} C_DIS
LIN {X 0.130,Y -403.643,Z 685.549,A 0.000,B 0.000,C 90.000,E1 134.757} C_DIS
LIN {X -0.214,Y -405.116,Z 685.545,A 0.000,B 0.000,C 90.000,E1 134.109} C_DIS
LIN {X 0.026,Y -407.822,Z 685.541,A 0.000,B 0.000,C 90.000,E1 133.380} C_DIS
LIN {X 0.165,Y -409.983,Z 685.539,A 0.000,B 0.000,C 90.000,E1 133.014} C_DIS
LIN {X 0.089,Y -411.287,Z 685.538,A 0.000,B 0.000,C 90.000,E1 132.852} C_DIS
LIN {X 0.037,Y -414.286,Z 685.536,A 0.000,B 0.000,C 90.000,E1 132.528} C_DIS
LIN {X -0.020,Y -427.587,Z 685.530,A 0.000,B 0.000,C 90.000,E1 131.310} C_DIS
LIN {X 0.054,Y -449.465,Z 685.519,A 0.000,B 0.000,C 90.000,E1 129.483} C_DIS
LIN {X -0.046,Y -461.887,Z 685.514,A 0.000,B 0.000,C 90.000,E1 128.508} C_DIS
LIN {X -0.094,Y -467.908,Z 685.511,A 0.000,B 0.000,C 90.000,E1 128.016} C_DIS
LIN {X 0.127,Y -476.751,Z 685.507,A 0.000,B 0.000,C 90.000,E1 127.237} C_DIS
LIN {X -0.191,Y -488.250,Z 685.501,A 0.000,B 0.000,C 90.000,E1 126.217} C_DIS
LIN {X -0.079,Y -492.497,Z 685.499,A 0.000,B 0.000,C 90.000,E1 125.804} C_DIS
LIN {X 0.141,Y -502.131,Z 685.494,A 0.000,B 0.000,C 90.000,E1 124.818} C_DIS
LIN {X 0.109,Y -508.838,Z 685.490,A 0.000,B 0.000,C 90.000,E1 124.119} C_DIS
LIN {X 0.120,Y -515.110,Z 685.486,A 0.000,B 0.000,C 90.000,E1 123.420} C_DIS
LIN {X -0.009,Y -521.241,Z 685.482,A 0.000,B 0.000,C 90.000,E1 122.704} C_DIS
LIN {X 0.043,Y -524.710,Z 685.479,A 0.000,B 0.000,C 90.000,E1 122.260} C_DIS
LIN {X -0.037,Y -529.906,Z 685.475,A 0.000,B 0.000,C 90.000,E1 121.544} C_DIS
LIN {X -0.223,Y -532.886,Z 685.473,A 0.000,B 0.000,C 90.000,E1 121.131} C_DIS
LIN {X -0.081,Y -536.482,Z 685.470,A 0.000,B 0.000,C 90.000,E1 120.541} C_DIS
LIN {X 0.064,Y -541.826,Z 685.464,A 0.000,B 0.000,C 90.000,E1 119.539} C_DIS
LIN {X -0.069,Y -544.066,Z 685.462,A 0.000,B 0.000,C 90.000,E1 119.127} C_DIS
LIN {X -0.092,Y -548.028,Z 685.457,A 0.000,B 0.000,C 90.000,E1 118.281} C_DIS
LIN {X -0.072,Y -551.740,Z 685.452,A 0.000,B 0.000,C 90.000,E1 117.436} C_DIS
LIN {X -0.044,Y -554.058,Z 685.449,A 0.000,B 0.000,C 90.000,E1 116.873} C_DIS
LIN {X 0.319,Y -558.293,Z 685.443,A 0.000,B 0.000,C 90.000,E1 115.720} C_DIS
LIN {X 0.199,Y -561.290,Z 685.438,A 0.000,B 0.000,C 90.000,E1 114.899} C_DIS
LIN {X 0.109,Y -564.010,Z 685.434,A 0.000,B 0.000,C 90.000,E1 114.079} C_DIS
LIN {X 0.046,Y -566.449,Z 685.429,A 0.000,B 0.000,C 90.000,E1 113.259} C_DIS
LIN {X -0.215,Y -568.617,Z 685.425,A 0.000,B 0.000,C 90.000,E1 112.461} C_DIS
LIN {X -0.099,Y -571.031,Z 685.419,A 0.000,B 0.000,C 90.000,E1 111.354} C_DIS
LIN {X 0.053,Y -573.236,Z 685.413,A 0.000,B 0.000,C 90.000,E1 110.248} C_DIS
LIN {X 0.231,Y -576.210,Z 685.404,A 0.000,B 0.000,C 90.000,E1 108.598} C_DIS
LIN {X 0.107,Y -579.195,Z 685.394,A 0.000,B 0.000,C 90.000,E1 106.985} C_DIS
LIN {X 0.171,Y -581.149,Z 685.388,A 0.000,B 0.000,C 90.000,E1 105.898} C_DIS
LIN {X -0.007,Y -583.867,Z 685.380,A 0.000,B 0.000,C 90.000,E1 104.300} C_DIS
LIN {X -0.135,Y -586.534,Z 685.371,A 0.000,B 0.000,C 90.000,E1 102.703} C_DIS
LIN {X 0.293,Y -588.315,Z 685.365,A 0.000,B 0.000,C 90.000,E1 101.591} C_DIS
LIN {X -0.260,Y -590.567,Z 685.357,A 0.000,B 0.000,C 90.000,E1 100.310} C_DIS
LIN {X -0.146,Y -591.844,Z 685.353,A 0.000,B 0.000,C 90.000,E1 99.500} C_DIS
LIN {X -0.055,Y -593.840,Z 685.345,A 0.000,B 0.000,C 90.000,E1 98.163} C_DIS
LIN {X 0.188,Y -596.078,Z 685.337,A 0.000,B 0.000,C 90.000,E1 96.549} C_DIS
LIN {X 0.262,Y -597.822,Z 685.329,A 0.000,B 0.000,C 90.000,E1 95.220} C_DIS
LIN {X -0.064,Y -599.782,Z 685.320,A 0.000,B 0.000,C 90.000,E1 93.669} C_DIS
LIN {X -0.029,Y -601.098,Z 685.313,A 0.000,B 0.000,C 90.000,E1 92.350} C_DIS
LIN {X 0.026,Y -602.247,Z 685.306,A 0.000,B 0.000,C 90.000,E1 91.031} C_DIS
LIN {X -0.166,Y -602.957,Z 685.300,A 0.000,B 0.000,C 90.000,E1 90.000} C_DIS
LIN {X -0.259,Y -603.309,Z 685.297,A 0.000,B 0.000,C 90.000,E1 89.484} C_DIS
LIN {X 0.090,Y -603.874,Z 685.288,A 0.000,B 0.000,C 90.000,E1 87.879} C_DIS
LIN {X -0.060,Y -604.133,Z 685.282,A 0.000,B 0.000,C 90.000,E1 86.846} C_DIS
LIN {X 0.045,Y -604.299,Z 685.275,A 0.000,B 0.000,C 90.000,E1 85.527} C_DIS
LIN {X 0.192,Y -604.262,Z 685.268,A 0.000,B 0.000,C 90.000,E1 84.204} C_DIS
LIN {X -0.198,Y -603.943,Z 685.261,A 0.000,B 0.000,C 90.000,E1 82.932} C_DIS
LIN {X 0.012,Y -603.462,Z 685.253,A 0.000,B 0.000,C 90.000,E1 81.602} C_DIS
LIN {X -0.013,Y -602.852,Z 685.248,A 0.000,B 0.000,C 90.000,E1 80.557} C_DIS
LIN {X 0.183,Y -601.301,Z 685.237,A 0.000,B 0.000,C 90.000,E1 78.701} C_DIS
LIN {X 0.255,Y -599.662,Z 685.229,A 0.000,B 0.000,C 90.000,E1 77.117} C_DIS
LIN {X -0.296,Y -598.487,Z 685.223,A 0.000,B 0.000,C 90.000,E1 76.117} C_DIS
LIN {X -0.141,Y -596.576,Z 685.214,A 0.000,B 0.000,C 90.000,E1 74.519} C_DIS
LIN {X -0.011,Y -595.114,Z 685.208,A 0.000,B 0.000,C 90.000,E1 73.449} C_DIS
LIN {X 0.271,Y -593.632,Z 685.202,A 0.000,B 0.000,C 90.000,E1 72.362} C_DIS
LIN {X -0.024,Y -592.046,Z 685.196,A 0.000,B 0.000,C 90.000,E1 71.329} C_DIS
LIN {X -0.222,Y -589.306,Z 685.187,A 0.000,B 0.000,C 90.000,E1 69.752} C_DIS
LIN {X -0.152,Y -586.753,Z 685.180,A 0.000,B 0.000,C 90.000,E1 68.411} C_DIS
LIN {X -0.330,Y -584.374,Z 685.174,A 0.000,B 0.000,C 90.000,E1 67.358} C_DIS
LIN {X 0.226,Y -581.742,Z 685.168,A 0.000,B 0.000,C 90.000,E1 66.230} C_DIS
LIN {X -0.027,Y -578.741,Z 685.162,A 0.000,B 0.000,C 90.000,E1 65.177} C_DIS
LIN {X 0.063,Y -576.333,Z 685.158,A 0.000,B 0.000,C 90.000,E1 64.357} C_DIS
LIN {X -0.134,Y -573.709,Z 685.153,A 0.000,B 0.000,C 90.000,E1 63.563} C_DIS
LIN {X -0.095,Y -570.935,Z 685.149,A 0.000,B 0.000,C 90.000,E1 62.743} C_DIS
LIN {X 0.171,Y -567.950,Z 685.144,A 0.000,B 0.000,C 90.000,E1 61.897} C_DIS
LIN {X -0.091,Y -564.762,Z 685.139,A 0.000,B 0.000,C 90.000,E1 61.101} C_DIS
LIN {X 0.110,Y -561.170,Z 685.135,A 0.000,B 0.000,C 90.000,E1 60.255} C_DIS
LIN {X -0.116,Y -557.952,Z 685.131,A 0.000,B 0.000,C 90.000,E1 59.587} C_DIS
LIN {X 0.107,Y -554.220,Z 685.127,A 0.000,B 0.000,C 90.000,E1 58.869} C_DIS
LIN {X -0.183,Y -550.035,Z 685.123,A 0.000,B 0.000,C 90.000,E1 58.201} C_DIS
LIN {X -0.323,Y -546.501,Z 685.120,A 0.000,B 0.000,C 90.000,E1 57.661} C_DIS
LIN {X 0.208,Y -542.601,Z 685.117,A 0.000,B 0.000,C 90.000,E1 57.041} C_DIS
LIN {X -0.043,Y -538.230,Z 685.114,A 0.000,B 0.000,C 90.000,E1 56.501} C_DIS
LIN {X -0.025,Y -533.403,Z 685.111,A 0.000,B 0.000,C 90.000,E1 55.928} C_DIS
LIN {X -0.187,Y -528.034,Z 685.108,A 0.000,B 0.000,C 90.000,E1 55.388} C_DIS
LIN {X -0.004,Y -522.193,Z 685.105,A 0.000,B 0.000,C 90.000,E1 54.848} C_DIS
LIN {X -0.061,Y -517.719,Z 685.103,A 0.000,B 0.000,C 90.000,E1 54.482} C_DIS
LIN {X 0.177,Y -511.307,Z 685.100,A 0.000,B 0.000,C 90.000,E1 53.989} C_DIS
LIN {X -0.163,Y -506.485,Z 685.098,A 0.000,B 0.000,C 90.000,E1 53.703} C_DIS
LIN {X 0.150,Y -499.868,Z 685.096,A 0.000,B 0.000,C 90.000,E1 53.256} C_DIS
LIN {X -0.077,Y -493.182,Z 685.094,A 0.000,B 0.000,C 90.000,E1 52.889} C_DIS
LIN {X 0.274,Y -481.472,Z 685.090,A 0.000,B 0.000,C 90.000,E1 52.190} C_DIS
LIN {X -0.011,Y -461.682,Z 685.084,A 0.000,B 0.000,C 90.000,E1 51.090} C_DIS
LIN {X -0.137,Y -445.531,Z 685.079,A 0.000,B 0.000,C 90.000,E1 50.150} C_DIS
LIN {X 0.004,Y -429.336,Z 685.073,A 0.000,B 0.000,C 90.000,E1 49.094} C_DIS
LIN {X -0.090,Y -426.892,Z 685.072,A 0.000,B 0.000,C 90.000,E1 48.933} C_DIS
LIN {X -0.115,Y -426.850,Z 685.072,A 0.000,B 0.000,C 90.000,E1 48.933} C_DIS
LIN {X -0.067,Y -418.653,Z 685.049,A 0.000,B 0.000,C 90.000,E1 44.838} C_DIS
LIN {X 0.036,Y -413.525,Z 685.037,A 0.000,B 0.000,C 90.000,E1 42.609} C_DIS
LIN {X -0.036,Y -413.375,Z 685.035,A 0.000,B 0.000,C 90.000,E1 42.285} C_DIS
LIN {X 0.051,Y -413.426,Z 685.023,A 0.000,B 0.000,C 90.000,E1 40.216} C_DIS
LIN {X -0.125,Y -414.095,Z 685.006,A 0.000,B 0.000,C 90.000,E1 37.156} C_DIS
LIN {X -0.075,Y -414.911,Z 684.997,A 0.000,B 0.000,C 90.000,E1 35.438} C_DIS
LIN {X 0.087,Y -415.670,Z 684.987,A 0.000,B 0.000,C 90.000,E1 33.706} C_DIS
LIN {X -0.014,Y -416.771,Z 684.976,A 0.000,B 0.000,C 90.000,E1 31.671} C_DIS
LIN {X 0.103,Y -417.681,Z 684.967,A 0.000,B 0.000,C 90.000,E1 29.951} C_DIS
LIN {X -0.049,Y -419.071,Z 684.953,A 0.000,B 0.000,C 90.000,E1 27.590} C_DIS
LIN {X 0.002,Y -420.712,Z 684.940,A 0.000,B 0.000,C 90.000,E1 25.207} C_DIS
LIN {X -0.143,Y -423.545,Z 684.921,A 0.000,B 0.000,C 90.000,E1 21.844} C_DIS
LIN {X 0.141,Y -425.171,Z 684.912,A 0.000,B 0.000,C 90.000,E1 20.120} C_DIS
LIN {X -0.097,Y -426.684,Z 684.903,A 0.000,B 0.000,C 90.000,E1 18.471} C_DIS
LIN {X -0.168,Y -428.236,Z 684.893,A 0.000,B 0.000,C 90.000,E1 16.804} C_DIS
LIN {X -0.099,Y -430.893,Z 684.878,A 0.000,B 0.000,C 90.000,E1 14.120} C_DIS
LIN {X -0.081,Y -433.097,Z 684.867,A 0.000,B 0.000,C 90.000,E1 12.119} C_DIS
LIN {X 0.083,Y -436.148,Z 684.853,A 0.000,B 0.000,C 90.000,E1 9.443} C_DIS
LIN {X -0.153,Y -439.461,Z 684.838,A 0.000,B 0.000,C 90.000,E1 6.834} C_DIS
LIN {X 0.165,Y -442.070,Z 684.827,A 0.000,B 0.000,C 90.000,E1 4.821} C_DIS
LIN {X 0.106,Y -444.935,Z 684.816,A 0.000,B 0.000,C 90.000,E1 2.865} C_DIS
LIN {X 0.000,Y -449.522,Z 684.800,A 0.000,B 0.000,C 90.000,E1 360.000} C_DIS
LIN {X -0.150,Y -455.128,Z 684.783,A 0.000,B 0.000,C 90.000,E1 356.906} C_DIS
LIN {X 0.099,Y -458.797,Z 684.772,A 0.000,B 0.000,C 90.000,E1 354.951} C_DIS
LIN {X -0.207,Y -461.850,Z 684.763,A 0.000,B 0.000,C 90.000,E1 353.394} C_DIS
LIN {X -0.002,Y -464.877,Z 684.754,A 0.000,B 0.000,C 90.000,E1 351.781} C_DIS
LIN {X -0.064,Y -467.873,Z 684.746,A 0.000,B 0.000,C 90.000,E1 350.208} C_DIS
LIN {X 0.119,Y -470.142,Z 684.739,A 0.000,B 0.000,C 90.000,E1 348.926} C_DIS
LIN {X -0.014,Y -473.495,Z 684.728,A 0.000,B 0.000,C 90.000,E1 347.061} C_DIS
LIN {X -0.069,Y -478.039,Z 684.714,A 0.000,B 0.000,C 90.000,E1 344.574} C_DIS
LIN {X 0.003,Y -481.030,Z 684.706,A 0.000,B 0.000,C 90.000,E1 343.015} C_DIS
LIN {X -0.006,Y -485.960,Z 684.692,A 0.000,B 0.000,C 90.000,E1 340.550} C_DIS
LIN {X -0.068,Y -489.712,Z 684.682,A 0.000,B 0.000,C 90.000,E1 338.720} C_DIS
LIN {X -0.285,Y -494.013,Z 684.670,A 0.000,B 0.000,C 90.000,E1 336.613} C_DIS
LIN {X 0.146,Y -497.123,Z 684.661,A 0.000,B 0.000,C 90.000,E1 335.049} C_DIS
LIN {X 0.013,Y -498.688,Z 684.658,A 0.000,B 0.000,C 90.000,E1 334.460} C_DIS
LIN {X 0.069,Y -499.558,Z 684.656,A 0.000,B 0.000,C 90.000,E1 334.152} C_DIS
LIN {X -0.069,Y -501.536,Z 684.654,A 0.000,B 0.000,C 90.000,E1 333.717} C_DIS
LIN {X 0.219,Y -503.280,Z 684.652,A 0.000,B 0.000,C 90.000,E1 333.384} C_DIS
LIN {X -0.162,Y -505.654,Z 684.651,A 0.000,B 0.000,C 90.000,E1 333.127} C_DIS
LIN {X 0.191,Y -510.672,Z 684.648,A 0.000,B 0.000,C 90.000,E1 332.615} C_DIS
LIN {X 0.236,Y -515.424,Z 684.646,A 0.000,B 0.000,C 90.000,E1 332.231} C_DIS
LIN {X -0.165,Y -530.516,Z 684.640,A 0.000,B 0.000,C 90.000,E1 331.257} C_DIS
LIN {X 0.184,Y -536.590,Z 684.638,A 0.000,B 0.000,C 90.000,E1 330.795} C_DIS
LIN {X -0.094,Y -542.504,Z 684.635,A 0.000,B 0.000,C 90.000,E1 330.383} C_DIS
LIN {X 0.018,Y -548.169,Z 684.633,A 0.000,B 0.000,C 90.000,E1 329.921} C_DIS
LIN {X -0.010,Y -556.488,Z 684.629,A 0.000,B 0.000,C 90.000,E1 329.203} C_DIS
LIN {X -0.086,Y -563.140,Z 684.625,A 0.000,B 0.000,C 90.000,E1 328.584} C_DIS
LIN {X 0.081,Y -571.027,Z 684.621,A 0.000,B 0.000,C 90.000,E1 327.788} C_DIS
LIN {X -0.079,Y -576.008,Z 684.618,A 0.000,B 0.000,C 90.000,E1 327.296} C_DIS
LIN {X 0.070,Y -584.613,Z 684.613,A 0.000,B 0.000,C 90.000,E1 326.373} C_DIS
LIN {X -0.167,Y -593.275,Z 684.608,A 0.000,B 0.000,C 90.000,E1 325.468} C_DIS
LIN {X -0.264,Y -600.481,Z 684.604,A 0.000,B 0.000,C 90.000,E1 324.689} C_DIS
LIN {X 0.228,Y -604.903,Z 684.601,A 0.000,B 0.000,C 90.000,E1 324.116} C_DIS
LIN {X -0.091,Y -609.168,Z 684.598,A 0.000,B 0.000,C 90.000,E1 323.623} C_DIS
LIN {X -0.095,Y -615.337,Z 684.594,A 0.000,B 0.000,C 90.000,E1 322.844} C_DIS
LIN {X -0.041,Y -620.899,Z 684.589,A 0.000,B 0.000,C 90.000,E1 322.065} C_DIS
LIN {X -0.034,Y -626.213,Z 684.585,A 0.000,B 0.000,C 90.000,E1 321.295} C_DIS
LIN {X 0.148,Y -630.372,Z 684.581,A 0.000,B 0.000,C 90.000,E1 320.642} C_DIS
LIN {X -0.142,Y -635.068,Z 684.577,A 0.000,B 0.000,C 90.000,E1 319.908} C_DIS
LIN {X 0.412,Y -641.089,Z 684.572,A 0.000,B 0.000,C 90.000,E1 318.852} C_DIS
LIN {X 0.083,Y -647.447,Z 684.565,A 0.000,B 0.000,C 90.000,E1 317.757} C_DIS
LIN {X -0.107,Y -652.174,Z 684.561,A 0.000,B 0.000,C 90.000,E1 316.905} C_DIS
LIN {X -0.246,Y -656.565,Z 684.556,A 0.000,B 0.000,C 90.000,E1 316.053} C_DIS
LIN {X 0.114,Y -660.651,Z 684.551,A 0.000,B 0.000,C 90.000,E1 315.162} C_DIS
LIN {X 0.059,Y -663.898,Z 684.547,A 0.000,B 0.000,C 90.000,E1 314.433} C_DIS
LIN {X 0.035,Y -670.148,Z 684.539,A 0.000,B 0.000,C 90.000,E1 312.975} C_DIS
LIN {X 0.139,Y -675.186,Z 684.532,A 0.000,B 0.000,C 90.000,E1 311.757} C_DIS
LIN {X -0.213,Y -678.931,Z 684.527,A 0.000,B 0.000,C 90.000,E1 310.825} C_DIS
LIN {X -0.042,Y -681.508,Z 684.523,A 0.000,B 0.000,C 90.000,E1 310.092} C_DIS
LIN {X 0.160,Y -683.876,Z 684.519,A 0.000,B 0.000,C 90.000,E1 309.358} C_DIS
LIN {X 0.007,Y -686.731,Z 684.513,A 0.000,B 0.000,C 90.000,E1 308.418} C_DIS
LIN {X 0.314,Y -689.302,Z 684.508,A 0.000,B 0.000,C 90.000,E1 307.443} C_DIS
LIN {X 0.225,Y -691.566,Z 684.503,A 0.000,B 0.000,C 90.000,E1 306.503} C_DIS
LIN {X 0.110,Y -693.115,Z 684.499,A 0.000,B 0.000,C 90.000,E1 305.804} C_DIS
LIN {X -0.339,Y -694.991,Z 684.494,A 0.000,B 0.000,C 90.000,E1 304.898} C_DIS
LIN {X 0.200,Y -696.599,Z 684.489,A 0.000,B 0.000,C 90.000,E1 303.913} C_DIS
LIN {X 0.372,Y -697.968,Z 684.483,A 0.000,B 0.000,C 90.000,E1 302.959} C_DIS
LIN {X -0.030,Y -699.148,Z 684.478,A 0.000,B 0.000,C 90.000,E1 302.054} C_DIS
LIN {X 0.065,Y -700.511,Z 684.472,A 0.000,B 0.000,C 90.000,E1 300.875} C_DIS
LIN {X -0.062,Y -701.450,Z 684.465,A 0.000,B 0.000,C 90.000,E1 299.716} C_DIS
LIN {X -0.262,Y -702.157,Z 684.459,A 0.000,B 0.000,C 90.000,E1 298.565} C_DIS
LIN {X 0.076,Y -703.461,Z 684.447,A 0.000,B 0.000,C 90.000,E1 296.437} C_DIS
LIN {X 0.297,Y -703.983,Z 684.443,A 0.000,B 0.000,C 90.000,E1 295.720} C_DIS
LIN {X -0.072,Y -703.839,Z 684.440,A 0.000,B 0.000,C 90.000,E1 295.283} C_DIS
LIN {X 0.213,Y -703.709,Z 684.439,A 0.000,B 0.000,C 90.000,E1 295.027} C_DIS
LIN {X -0.142,Y -703.112,Z 684.438,A 0.000,B 0.000,C 90.000,E1 294.823} C_DIS
LIN {X 0.127,Y -701.511,Z 684.435,A 0.000,B 0.000,C 90.000,E1 294.335} C_DIS
LIN {X 0.266,Y -700.803,Z 684.435,A 0.000,B 0.000,C 90.000,E1 294.207} C_DIS
LIN {X -0.100,Y -698.645,Z 684.433,A 0.000,B 0.000,C 90.000,E1 294.003} C_DIS
LIN {X 0.101,Y -694.929,Z 684.431,A 0.000,B 0.000,C 90.000,E1 293.643} C_DIS
LIN {X 0.308,Y -692.991,Z 684.431,A 0.000,B 0.000,C 90.000,E1 293.515} C_DIS
LIN {X -0.268,Y -688.345,Z 684.430,A 0.000,B 0.000,C 90.000,E1 293.387} C_DIS
LIN {X 0.046,Y -682.027,Z 684.429,A 0.000,B 0.000,C 90.000,E1 293.206} C_DIS
LIN {X 0.172,Y -679.903,Z 684.429,A 0.000,B 0.000,C 90.000,E1 293.153} C_DIS
LIN {X -0.203,Y -667.075,Z 684.428,A 0.000,B 0.000,C 90.000,E1 293.025} C_DIS
LIN {X 0.244,Y -655.021,Z 684.427,A 0.000,B 0.000,C 90.000,E1 292.823} C_DIS
LIN {X -0.186,Y -644.973,Z 684.426,A 0.000,B 0.000,C 90.000,E1 292.695} C_DIS
LIN {X 0.012,Y -631.703,Z 684.425,A 0.000,B 0.000,C 90.000,E1 292.408} C_DIS
LIN {X 0.030,Y -618.420,Z 684.423,A 0.000,B 0.000,C 90.000,E1 292.078} C_DIS
LIN {X -0.228,Y -594.425,Z 684.419,A 0.000,B 0.000,C 90.000,E1 291.408} C_DIS
LIN {X -0.018,Y -575.162,Z 684.416,A 0.000,B 0.000,C 90.000,E1 290.791} C_DIS
LIN {X 0.012,Y -562.789,Z 684.414,A 0.000,B 0.000,C 90.000,E1 290.429} C_DIS
LIN {X -0.156,Y -556.952,Z 684.412,A 0.000,B 0.000,C 90.000,E1 290.174} C_DIS
LIN {X 0.049,Y -555.482,Z 684.411,A 0.000,B 0.000,C 90.000,E1 289.993} C_DIS
LIN {X 0.007,Y -555.458,Z 684.411,A 0.000,B 0.000,C 90.000,E1 289.993} C_DIS
LIN {X 0.264,Y -554.614,Z 684.409,A 0.000,B 0.000,C 90.000,E1 289.631} C_DIS
LIN {X 0.005,Y -554.176,Z 684.405,A 0.000,B 0.000,C 90.000,E1 288.960} C_DIS
LIN {X -0.173,Y -553.775,Z 684.398,A 0.000,B 0.000,C 90.000,E1 287.583} C_DIS
LIN {X 0.030,Y -553.162,Z 684.387,A 0.000,B 0.000,C 90.000,E1 285.607} C_DIS
LIN {X -0.309,Y -552.619,Z 684.379,A 0.000,B 0.000,C 90.000,E1 284.245} C_DIS
LIN {X -0.243,Y -552.154,Z 684.373,A 0.000,B 0.000,C 90.000,E1 283.119} C_DIS
LIN {X -0.193,Y -551.442,Z 684.365,A 0.000,B 0.000,C 90.000,E1 281.715} C_DIS
LIN {X -0.156,Y -550.754,Z 684.357,A 0.000,B 0.000,C 90.000,E1 280.310} C_DIS
LIN {X 0.009,Y -549.852,Z 684.345,A 0.000,B 0.000,C 90.000,E1 278.049} C_DIS
LIN {X -0.060,Y -549.461,Z 684.335,A 0.000,B 0.000,C 90.000,E1 276.372} C_DIS
LIN {X -0.205,Y -549.229,Z 684.326,A 0.000,B 0.000,C 90.000,E1 274.702} C_DIS
LIN {X 0.067,Y -549.145,Z 684.318,A 0.000,B 0.000,C 90.000,E1 273.269} C_DIS
LIN {X -0.202,Y -548.887,Z 684.310,A 0.000,B 0.000,C 90.000,E1 271.892} C_DIS
LIN {X 0.069,Y -548.309,Z 684.303,A 0.000,B 0.000,C 90.000,E1 270.458} C_DIS
LIN {X -0.143,Y -547.164,Z 684.292,A 0.000,B 0.000,C 90.000,E1 268.511} C_DIS
LIN {X 0.090,Y -546.349,Z 684.284,A 0.000,B 0.000,C 90.000,E1 267.078} C_DIS
LIN {X -0.204,Y -545.322,Z 684.276,A 0.000,B 0.000,C 90.000,E1 265.698} C_DIS
LIN {X 0.008,Y -544.516,Z 684.270,A 0.000,B 0.000,C 90.000,E1 264.546} C_DIS
LIN {X 0.208,Y -543.637,Z 684.263,A 0.000,B 0.000,C 90.000,E1 263.394} C_DIS
LIN {X -0.070,Y -542.147,Z 684.256,A 0.000,B 0.000,C 90.000,E1 262.008} C_DIS
LIN {X -0.016,Y -539.385,Z 684.240,A 0.000,B 0.000,C 90.000,E1 259.162} C_DIS
LIN {X -0.125,Y -537.916,Z 684.230,A 0.000,B 0.000,C 90.000,E1 257.465} C_DIS
LIN {X -0.147,Y -536.501,Z 684.221,A 0.000,B 0.000,C 90.000,E1 255.755} C_DIS
LIN {X -0.257,Y -535.158,Z 684.213,A 0.000,B 0.000,C 90.000,E1 254.338} C_DIS
LIN {X -0.027,Y -533.110,Z 684.202,A 0.000,B 0.000,C 90.000,E1 252.308} C_DIS
LIN {X -0.022,Y -531.125,Z 684.191,A 0.000,B 0.000,C 90.000,E1 250.296} C_DIS
LIN {X 0.058,Y -529.326,Z 684.183,A 0.000,B 0.000,C 90.000,E1 248.847} C_DIS
LIN {X -0.188,Y -527.692,Z 684.176,A 0.000,B 0.000,C 90.000,E1 247.720} C_DIS
LIN {X 0.209,Y -525.588,Z 684.168,A 0.000,B 0.000,C 90.000,E1 246.230} C_DIS
LIN {X -0.240,Y -522.658,Z 684.158,A 0.000,B 0.000,C 90.000,E1 244.537} C_DIS
LIN {X -0.029,Y -521.100,Z 684.154,A 0.000,B 0.000,C 90.000,E1 243.640} C_DIS
LIN {X -0.122,Y -517.655,Z 684.144,A 0.000,B 0.000,C 90.000,E1 241.897} C_DIS
LIN {X 0.044,Y -514.724,Z 684.136,A 0.000,B 0.000,C 90.000,E1 240.411} C_DIS
LIN {X -0.137,Y -510.943,Z 684.126,A 0.000,B 0.000,C 90.000,E1 238.663} C_DIS
LIN {X 0.079,Y -508.361,Z 684.119,A 0.000,B 0.000,C 90.000,E1 237.454} C_DIS
LIN {X 0.033,Y -504.304,Z 684.109,A 0.000,B 0.000,C 90.000,E1 235.674} C_DIS
LIN {X 0.001,Y -501.499,Z 684.103,A 0.000,B 0.000,C 90.000,E1 234.482} C_DIS
LIN {X 0.101,Y -497.825,Z 684.094,A 0.000,B 0.000,C 90.000,E1 232.970} C_DIS
LIN {X -0.008,Y -493.410,Z 684.084,A 0.000,B 0.000,C 90.000,E1 231.170} C_DIS
LIN {X -0.133,Y -489.727,Z 684.076,A 0.000,B 0.000,C 90.000,E1 229.666} C_DIS
LIN {X -0.030,Y -484.691,Z 684.064,A 0.000,B 0.000,C 90.000,E1 227.514} C_DIS
LIN {X 0.132,Y -480.376,Z 684.054,A 0.000,B 0.000,C 90.000,E1 225.648} C_DIS
LIN {X -0.170,Y -478.267,Z 684.049,A 0.000,B 0.000,C 90.000,E1 224.757} C_DIS
LIN {X 0.268,Y -473.205,Z 684.036,A 0.000,B 0.000,C 90.000,E1 222.528} C_DIS
LIN {X -0.307,Y -467.764,Z 684.023,A 0.000,B 0.000,C 90.000,E1 220.092} C_DIS
LIN {X -0.125,Y -463.727,Z 684.012,A 0.000,B 0.000,C 90.000,E1 218.177} C_DIS
LIN {X 0.017,Y -456.919,Z 683.993,A 0.000,B 0.000,C 90.000,E1 214.659} C_DIS
LIN {X 0.160,Y -453.861,Z 683.984,A 0.000,B 0.000,C 90.000,E1 213.038} C_DIS
LIN {X -0.041,Y -450.159,Z 683.973,A 0.000,B 0.000,C 90.000,E1 211.131} C_DIS
LIN {X -0.180,Y -446.486,Z 683.962,A 0.000,B 0.000,C 90.000,E1 209.205} C_DIS
LIN {X -0.135,Y -444.140,Z 683.955,A 0.000,B 0.000,C 90.000,E1 207.897} C_DIS
LIN {X 0.106,Y -441.205,Z 683.946,A 0.000,B 0.000,C 90.000,E1 206.232} C_DIS
LIN {X 0.120,Y -437.679,Z 683.935,A 0.000,B 0.000,C 90.000,E1 204.259} C_DIS
LIN {X 0.035,Y -435.240,Z 683.928,A 0.000,B 0.000,C 90.000,E1 202.950} C_DIS
LIN {X 0.134,Y -432.220,Z 683.918,A 0.000,B 0.000,C 90.000,E1 201.280} C_DIS
LIN {X -0.175,Y -428.556,Z 683.907,A 0.000,B 0.000,C 90.000,E1 199.322} C_DIS
LIN {X 0.099,Y -424.993,Z 683.896,A 0.000,B 0.000,C 90.000,E1 197.275} C_DIS
LIN {X -0.081,Y -422.717,Z 683.889,A 0.000,B 0.000,C 90.000,E1 195.953} C_DIS
LIN {X 0.055,Y -419.806,Z 683.879,A 0.000,B 0.000,C 90.000,E1 194.245} C_DIS
LIN {X 0.026,Y -414.575,Z 683.862,A 0.000,B 0.000,C 90.000,E1 191.186} C_DIS
LIN {X -0.161,Y -411.874,Z 683.853,A 0.000,B 0.000,C 90.000,E1 189.500} C_DIS
LIN {X 0.033,Y -407.173,Z 683.835,A 0.000,B 0.000,C 90.000,E1 186.372} C_DIS
LIN {X -0.083,Y -403.319,Z 683.820,A 0.000,B 0.000,C 90.000,E1 183.612} C_DIS
LIN {X 0.036,Y -399.930,Z 683.805,A 0.000,B 0.000,C 90.000,E1 180.802} C_DIS
LIN {X 0.193,Y -398.172,Z 683.795,A 0.000,B 0.000,C 90.000,E1 179.026} C_DIS
LIN {X 0.042,Y -395.288,Z 683.775,A 0.000,B 0.000,C 90.000,E1 175.527} C_DIS
LIN {X 0.002,Y -393.659,Z 683.760,A 0.000,B 0.000,C 90.000,E1 172.704} C_DIS
LIN {X 0.114,Y -392.755,Z 683.746,A 0.000,B 0.000,C 90.000,E1 170.208} C_DIS
LIN {X -0.109,Y -392.331,Z 683.732,A 0.000,B 0.000,C 90.000,E1 167.757} C_DIS
LIN {X -0.165,Y -392.116,Z 683.726,A 0.000,B 0.000,C 90.000,E1 166.700} C_DIS
LIN {X -0.163,Y -391.779,Z 683.708,A 0.000,B 0.000,C 90.000,E1 163.504} C_DIS
LIN {X 0.227,Y -391.782,Z 683.693,A 0.000,B 0.000,C 90.000,E1 160.604} C_DIS
LIN {X -0.081,Y -391.909,Z 683.681,A 0.000,B 0.000,C 90.000,E1 158.518} C_DIS
LIN {X -0.002,Y -392.207,Z 683.665,A 0.000,B 0.000,C 90.000,E1 155.665} C_DIS
LIN {X 0.159,Y -392.392,Z 683.653,A 0.000,B 0.000,C 90.000,E1 153.512} C_DIS
LIN {X 0.144,Y -392.833,Z 683.641,A 0.000,B 0.000,C 90.000,E1 151.385} C_DIS
LIN {X 0.119,Y -393.278,Z 683.631,A 0.000,B 0.000,C 90.000,E1 149.616} C_DIS
LIN {X 0.034,Y -393.927,Z 683.620,A 0.000,B 0.000,C 90.000,E1 147.502} C_DIS
LIN {X 0.111,Y -394.710,Z 683.610,A 0.000,B 0.000,C 90.000,E1 145.722} C_DIS
LIN {X 0.012,Y -396.546,Z 683.592,A 0.000,B 0.000,C 90.000,E1 142.557} C_DIS
LIN {X 0.169,Y -398.358,Z 683.578,A 0.000,B 0.000,C 90.000,E1 140.070} C_DIS
LIN {X 0.101,Y -399.839,Z 683.569,A 0.000,B 0.000,C 90.000,E1 138.324} C_DIS
LIN {X 0.184,Y -402.909,Z 683.551,A 0.000,B 0.000,C 90.000,E1 135.162} C_DIS
LIN {X -0.164,Y -403.951,Z 683.547,A 0.000,B 0.000,C 90.000,E1 134.514} C_DIS
LIN {X 0.151,Y -404.967,Z 683.544,A 0.000,B 0.000,C 90.000,E1 133.947} C_DIS
LIN {X -0.001,Y -406.325,Z 683.542,A 0.000,B 0.000,C 90.000,E1 133.623} C_DIS
LIN {X -0.165,Y -407.489,Z 683.540,A 0.000,B 0.000,C 90.000,E1 133.299} C_DIS
LIN {X -0.033,Y -409.185,Z 683.539,A 0.000,B 0.000,C 90.000,E1 133.014} C_DIS
LIN {X -0.112,Y -410.131,Z 683.538,A 0.000,B 0.000,C 90.000,E1 132.852} C_DIS
LIN {X -0.189,Y -411.358,Z 683.537,A 0.000,B 0.000,C 90.000,E1 132.690} C_DIS
LIN {X -0.050,Y -415.341,Z 683.535,A 0.000,B 0.000,C 90.000,E1 132.243} C_DIS
LIN {X 0.052,Y -427.305,Z 683.529,A 0.000,B 0.000,C 90.000,E1 131.148} C_DIS
LIN {X -0.088,Y -449.221,Z 683.519,A 0.000,B 0.000,C 90.000,E1 129.358} C_DIS
LIN {X -0.162,Y -461.657,Z 683.513,A 0.000,B 0.000,C 90.000,E1 128.382} C_DIS
LIN {X 0.082,Y -469.221,Z 683.510,A 0.000,B 0.000,C 90.000,E1 127.729} C_DIS
LIN {X 0.212,Y -476.680,Z 683.506,A 0.000,B 0.000,C 90.000,E1 127.076} C_DIS
LIN {X 0.051,Y -486.406,Z 683.501,A 0.000,B 0.000,C 90.000,E1 126.217} C_DIS
LIN {X -0.193,Y -491.968,Z 683.498,A 0.000,B 0.000,C 90.000,E1 125.724} C_DIS
LIN {X -0.135,Y -500.334,Z 683.494,A 0.000,B 0.000,C 90.000,E1 124.898} C_DIS
LIN {X -0.120,Y -507.089,Z 683.490,A 0.000,B 0.000,C 90.000,E1 124.199} C_DIS
LIN {X -0.220,Y -511.056,Z 683.488,A 0.000,B 0.000,C 90.000,E1 123.785} C_DIS
LIN {X 0.173,Y -516.179,Z 683.484,A 0.000,B 0.000,C 90.000,E1 123.166} C_DIS
LIN {X -0.132,Y -519.671,Z 683.482,A 0.000,B 0.000,C 90.000,E1 122.801} C_DIS
LIN {X 0.023,Y -524.260,Z 683.479,A 0.000,B 0.000,C 90.000,E1 122.212} C_DIS
LIN {X 0.152,Y -528.275,Z 683.476,A 0.000,B 0.000,C 90.000,E1 121.671} C_DIS
LIN {X -0.071,Y -532.233,Z 683.473,A 0.000,B 0.000,C 90.000,E1 121.131} C_DIS
LIN {X 0.118,Y -536.689,Z 683.469,A 0.000,B 0.000,C 90.000,E1 120.413} C_DIS
LIN {X -0.045,Y -540.696,Z 683.465,A 0.000,B 0.000,C 90.000,E1 119.716} C_DIS
LIN {X 0.026,Y -544.423,Z 683.461,A 0.000,B 0.000,C 90.000,E1 118.999} C_DIS
LIN {X 0.010,Y -548.392,Z 683.456,A 0.000,B 0.000,C 90.000,E1 118.153} C_DIS
LIN {X -0.104,Y -551.551,Z 683.453,A 0.000,B 0.000,C 90.000,E1 117.462} C_DIS
LIN {X -0.044,Y -554.996,Z 683.448,A 0.000,B 0.000,C 90.000,E1 116.616} C_DIS
LIN {X 0.042,Y -558.202,Z 683.443,A 0.000,B 0.000,C 90.000,E1 115.771} C_DIS
LIN {X -0.084,Y -561.254,Z 683.439,A 0.000,B 0.000,C 90.000,E1 114.951} C_DIS
LIN {X 0.141,Y -564.886,Z 683.432,A 0.000,B 0.000,C 90.000,E1 113.823} C_DIS
LIN {X -0.138,Y -567.235,Z 683.428,A 0.000,B 0.000,C 90.000,E1 113.025} C_DIS
LIN {X -0.170,Y -569.327,Z 683.423,A 0.000,B 0.000,C 90.000,E1 112.206} C_DIS
LIN {X 0.133,Y -571.168,Z 683.419,A 0.000,B 0.000,C 90.000,E1 111.354} C_DIS
LIN {X -0.072,Y -572.858,Z 683.414,A 0.000,B 0.000,C 90.000,E1 110.556} C_DIS
LIN {X -0.265,Y -575.424,Z 683.407,A 0.000,B 0.000,C 90.000,E1 109.214} C_DIS
LIN {X -0.227,Y -578.447,Z 683.398,A 0.000,B 0.000,C 90.000,E1 107.583} C_DIS
LIN {X 0.043,Y -580.957,Z 683.390,A 0.000,B 0.000,C 90.000,E1 106.205} C_DIS
LIN {X 0.350,Y -583.293,Z 683.383,A 0.000,B 0.000,C 90.000,E1 104.828} C_DIS
LIN {X 0.077,Y -586.004,Z 683.374,A 0.000,B 0.000,C 90.000,E1 103.244} C_DIS
LIN {X 0.189,Y -588.260,Z 683.366,A 0.000,B 0.000,C 90.000,E1 101.895} C_DIS
LIN {X 0.020,Y -590.971,Z 683.357,A 0.000,B 0.000,C 90.000,E1 100.310} C_DIS
LIN {X -0.175,Y -592.707,Z 683.351,A 0.000,B 0.000,C 90.000,E1 99.265} C_DIS
LIN {X 0.240,Y -594.317,Z 683.346,A 0.000,B 0.000,C 90.000,E1 98.163} C_DIS
LIN {X -0.099,Y -596.594,Z 683.337,A 0.000,B 0.000,C 90.000,E1 96.606} C_DIS
LIN {X 0.207,Y -598.714,Z 683.328,A 0.000,B 0.000,C 90.000,E1 94.992} C_DIS
LIN {X 0.264,Y -600.333,Z 683.321,A 0.000,B 0.000,C 90.000,E1 93.669} C_DIS
LIN {X 0.064,Y -601.439,Z 683.315,A 0.000,B 0.000,C 90.000,E1 92.636} C_DIS
LIN {X 0.124,Y -602.635,Z 683.307,A 0.000,B 0.000,C 90.000,E1 91.318} C_DIS
LIN {X -0.065,Y -603.438,Z 683.302,A 0.000,B 0.000,C 90.000,E1 90.286} C_DIS
LIN {X -0.243,Y -604.037,Z 683.296,A 0.000,B 0.000,C 90.000,E1 89.255} C_DIS
LIN {X 0.206,Y -604.408,Z 683.290,A 0.000,B 0.000,C 90.000,E1 88.165} C_DIS
LIN {X -0.312,Y -604.784,Z 683.283,A 0.000,B 0.000,C 90.000,E1 86.906} C_DIS
LIN {X -0.162,Y -604.886,Z 683.275,A 0.000,B 0.000,C 90.000,E1 85.584} C_DIS
LIN {X -0.254,Y -604.851,Z 683.270,A 0.000,B 0.000,C 90.000,E1 84.546} C_DIS
LIN {X -0.050,Y -604.752,Z 683.265,A 0.000,B 0.000,C 90.000,E1 83.742} C_DIS
LIN {X 0.171,Y -604.379,Z 683.258,A 0.000,B 0.000,C 90.000,E1 82.413} C_DIS
LIN {X 0.067,Y -603.929,Z 683.252,A 0.000,B 0.000,C 90.000,E1 81.376} C_DIS
LIN {X 0.042,Y -603.214,Z 683.246,A 0.000,B 0.000,C 90.000,E1 80.330} C_DIS
LIN {X 0.038,Y -601.839,Z 683.238,A 0.000,B 0.000,C 90.000,E1 78.757} C_DIS
LIN {X 0.126,Y -600.152,Z 683.229,A 0.000,B 0.000,C 90.000,E1 77.173} C_DIS
LIN {X 0.164,Y -598.954,Z 683.223,A 0.000,B 0.000,C 90.000,E1 76.117} C_DIS
LIN {X -0.248,Y -597.012,Z 683.214,A 0.000,B 0.000,C 90.000,E1 74.574} C_DIS
LIN {X 0.337,Y -595.143,Z 683.207,A 0.000,B 0.000,C 90.000,E1 73.196} C_DIS
LIN {X -0.120,Y -593.593,Z 683.201,A 0.000,B 0.000,C 90.000,E1 72.181} C_DIS
LIN {X 0.147,Y -591.923,Z 683.195,A 0.000,B 0.000,C 90.000,E1 71.094} C_DIS
LIN {X 0.264,Y -589.610,Z 683.188,A 0.000,B 0.000,C 90.000,E1 69.752} C_DIS
LIN {X -0.209,Y -587.014,Z 683.180,A 0.000,B 0.000,C 90.000,E1 68.465} C_DIS
LIN {X 0.161,Y -584.586,Z 683.174,A 0.000,B 0.000,C 90.000,E1 67.358} C_DIS
LIN {X -0.049,Y -581.920,Z 683.168,A 0.000,B 0.000,C 90.000,E1 66.305} C_DIS
LIN {X -0.062,Y -578.863,Z 683.162,A 0.000,B 0.000,C 90.000,E1 65.229} C_DIS
LIN {X 0.033,Y -576.411,Z 683.158,A 0.000,B 0.000,C 90.000,E1 64.409} C_DIS
LIN {X 0.099,Y -573.753,Z 683.153,A 0.000,B 0.000,C 90.000,E1 63.589} C_DIS
LIN {X 0.226,Y -569.910,Z 683.147,A 0.000,B 0.000,C 90.000,E1 62.487} C_DIS
LIN {X -0.114,Y -567.905,Z 683.144,A 0.000,B 0.000,C 90.000,E1 61.975} C_DIS
LIN {X 0.116,Y -564.647,Z 683.140,A 0.000,B 0.000,C 90.000,E1 61.129} C_DIS
LIN {X -0.279,Y -560.324,Z 683.134,A 0.000,B 0.000,C 90.000,E1 60.205} C_DIS
LIN {X 0.073,Y -557.695,Z 683.131,A 0.000,B 0.000,C 90.000,E1 59.616} C_DIS
LIN {X -0.188,Y -553.893,Z 683.127,A 0.000,B 0.000,C 90.000,E1 58.948} C_DIS
LIN {X 0.277,Y -549.628,Z 683.124,A 0.000,B 0.000,C 90.000,E1 58.201} C_DIS
LIN {X 0.073,Y -545.964,Z 683.120,A 0.000,B 0.000,C 90.000,E1 57.661} C_DIS
LIN {X -0.152,Y -541.980,Z 683.117,A 0.000,B 0.000,C 90.000,E1 57.120} C_DIS
LIN {X -0.110,Y -537.497,Z 683.114,A 0.000,B 0.000,C 90.000,E1 56.548} C_DIS
LIN {X 0.116,Y -532.493,Z 683.111,A 0.000,B 0.000,C 90.000,E1 55.960} C_DIS
LIN {X -0.108,Y -527.409,Z 683.108,A 0.000,B 0.000,C 90.000,E1 55.468} C_DIS
LIN {X 0.102,Y -521.966,Z 683.106,A 0.000,B 0.000,C 90.000,E1 54.975} C_DIS
LIN {X -0.253,Y -518.024,Z 683.104,A 0.000,B 0.000,C 90.000,E1 54.689} C_DIS
LIN {X 0.089,Y -511.828,Z 683.101,A 0.000,B 0.000,C 90.000,E1 54.196} C_DIS
LIN {X -0.139,Y -505.161,Z 683.099,A 0.000,B 0.000,C 90.000,E1 53.783} C_DIS
LIN {X 0.214,Y -498.462,Z 683.096,A 0.000,B 0.000,C 90.000,E1 53.336} C_DIS
LIN {X 0.116,Y -491.922,Z 683.094,A 0.000,B 0.000,C 90.000,E1 52.970} C_DIS
LIN {X -0.216,Y -478.708,Z 683.090,A 0.000,B 0.000,C 90.000,E1 52.271} C_DIS
LIN {X -0.041,Y -460.656,Z 683.085,A 0.000,B 0.000,C 90.000,E1 51.215} C_DIS
LIN {X 0.051,Y -446.245,Z 683.080,A 0.000,B 0.000,C 90.000,E1 50.356} C_DIS
LIN {X -0.059,Y -433.081,Z 683.075,A 0.000,B 0.000,C 90.000,E1 49.542} C_DIS
LIN {X 0.038,Y -427.397,Z 683.073,A 0.000,B 0.000,C 90.000,E1 49.138} C_DIS
LIN {X 0.012,Y -427.368,Z 683.073,A 0.000,B 0.000,C 90.000,E1 49.138} C_DIS
LIN {X 0.053,Y -418.414,Z 683.049,A 0.000,B 0.000,C 90.000,E1 44.717} C_DIS
LIN {X -0.044,Y -413.852,Z 683.038,A 0.000,B 0.000,C 90.000,E1 42.771} C_DIS
LIN {X -0.090,Y -413.865,Z 683.025,A 0.000,B 0.000,C 90.000,E1 40.539} C_DIS
LIN {X 0.012,Y -414.484,Z 683.008,A 0.000,B 0.000,C 90.000,E1 37.443} C_DIS
LIN {X 0.006,Y -415.409,Z 682.997,A 0.000,B 0.000,C 90.000,E1 35.391} C_DIS
LIN {X -0.160,Y -416.180,Z 682.987,A 0.000,B 0.000,C 90.000,E1 33.706} C_DIS
LIN {X -0.249,Y -417.298,Z 682.976,A 0.000,B 0.000,C 90.000,E1 31.671} C_DIS
LIN {X 0.087,Y -418.207,Z 682.966,A 0.000,B 0.000,C 90.000,E1 29.922} C_DIS
LIN {X -0.066,Y -419.616,Z 682.953,A 0.000,B 0.000,C 90.000,E1 27.564} C_DIS
LIN {X 0.187,Y -421.216,Z 682.940,A 0.000,B 0.000,C 90.000,E1 25.155} C_DIS
LIN {X 0.073,Y -424.096,Z 682.921,A 0.000,B 0.000,C 90.000,E1 21.791} C_DIS
LIN {X -0.025,Y -425.714,Z 682.912,A 0.000,B 0.000,C 90.000,E1 20.120} C_DIS
LIN {X -0.047,Y -426.947,Z 682.904,A 0.000,B 0.000,C 90.000,E1 18.779} C_DIS
LIN {X 0.219,Y -428.695,Z 682.893,A 0.000,B 0.000,C 90.000,E1 16.732} C_DIS
LIN {X -0.025,Y -430.953,Z 682.880,A 0.000,B 0.000,C 90.000,E1 14.426} C_DIS
LIN {X 0.099,Y -433.094,Z 682.869,A 0.000,B 0.000,C 90.000,E1 12.411} C_DIS
LIN {X 0.128,Y -435.703,Z 682.856,A 0.000,B 0.000,C 90.000,E1 10.084} C_DIS
LIN {X -0.199,Y -438.486,Z 682.843,A 0.000,B 0.000,C 90.000,E1 7.814} C_DIS
LIN {X 0.136,Y -441.052,Z 682.832,A 0.000,B 0.000,C 90.000,E1 5.796} C_DIS
LIN {X 0.013,Y -445.186,Z 682.816,A 0.000,B 0.000,C 90.000,E1 2.865} C_DIS
LIN {X 0.000,Y -449.731,Z 682.800,A 0.000,B 0.000,C 90.000,E1 360.000} C_DIS
LIN {X -0.143,Y -455.295,Z 682.783,A 0.000,B 0.000,C 90.000,E1 356.906} C_DIS
LIN {X 0.111,Y -458.946,Z 682.772,A 0.000,B 0.000,C 90.000,E1 354.951} C_DIS
LIN {X -0.005,Y -462.599,Z 682.761,A 0.000,B 0.000,C 90.000,E1 353.053} C_DIS
LIN {X -0.188,Y -465.601,Z 682.753,A 0.000,B 0.000,C 90.000,E1 351.489} C_DIS
LIN {X -0.044,Y -467.991,Z 682.746,A 0.000,B 0.000,C 90.000,E1 350.208} C_DIS
LIN {X 0.140,Y -470.263,Z 682.739,A 0.000,B 0.000,C 90.000,E1 348.926} C_DIS
LIN {X -0.054,Y -474.147,Z 682.726,A 0.000,B 0.000,C 90.000,E1 346.756} C_DIS
LIN {X -0.042,Y -478.152,Z 682.714,A 0.000,B 0.000,C 90.000,E1 344.574} C_DIS
LIN {X 0.032,Y -481.140,Z 682.706,A 0.000,B 0.000,C 90.000,E1 343.015} C_DIS
LIN {X 0.027,Y -486.052,Z 682.692,A 0.000,B 0.000,C 90.000,E1 340.550} C_DIS
LIN {X -0.006,Y -490.432,Z 682.680,A 0.000,B 0.000,C 90.000,E1 338.411} C_DIS
LIN {X -0.247,Y -494.085,Z 682.670,A 0.000,B 0.000,C 90.000,E1 336.613} C_DIS
LIN {X -0.214,Y -497.755,Z 682.660,A 0.000,B 0.000,C 90.000,E1 334.793} C_DIS
LIN {X -0.089,Y -499.742,Z 682.656,A 0.000,B 0.000,C 90.000,E1 334.024} C_DIS
LIN {X -0.176,Y -501.756,Z 682.653,A 0.000,B 0.000,C 90.000,E1 333.512} C_DIS
LIN {X -0.113,Y -503.402,Z 682.651,A 0.000,B 0.000,C 90.000,E1 333.204} C_DIS
LIN {X -0.101,Y -507.048,Z 682.649,A 0.000,B 0.000,C 90.000,E1 332.743} C_DIS
LIN {X 0.069,Y -511.525,Z 682.646,A 0.000,B 0.000,C 90.000,E1 332.308} C_DIS
LIN {X -0.175,Y -515.293,Z 682.645,A 0.000,B 0.000,C 90.000,E1 332.025} C_DIS
LIN {X 0.033,Y -527.531,Z 682.640,A 0.000,B 0.000,C 90.000,E1 331.179} C_DIS
LIN {X -0.230,Y -538.244,Z 682.636,A 0.000,B 0.000,C 90.000,E1 330.461} C_DIS
LIN {X 0.071,Y -545.446,Z 682.633,A 0.000,B 0.000,C 90.000,E1 329.871} C_DIS
LIN {X 0.000,Y -551.114,Z 682.630,A 0.000,B 0.000,C 90.000,E1 329.410} C_DIS
LIN {X 0.044,Y -556.632,Z 682.627,A 0.000,B 0.000,C 90.000,E1 328.918} C_DIS
LIN {X 0.136,Y -560.668,Z 682.625,A 0.000,B 0.000,C 90.000,E1 328.535} C_DIS
LIN {X -0.128,Y -569.920,Z 682.620,A 0.000,B 0.000,C 90.000,E1 327.661} C_DIS
LIN {X 0.054,Y -576.292,Z 682.617,A 0.000,B 0.000,C 90.000,E1 326.993} C_DIS
LIN {X -0.063,Y -583.823,Z 682.612,A 0.000,B 0.000,C 90.000,E1 326.215} C_DIS
LIN {X -0.104,Y -593.605,Z 682.607,A 0.000,B 0.000,C 90.000,E1 325.182} C_DIS
LIN {X 0.035,Y -598.513,Z 682.604,A 0.000,B 0.000,C 90.000,E1 324.642} C_DIS
LIN {X -0.052,Y -605.245,Z 682.599,A 0.000,B 0.000,C 90.000,E1 323.863} C_DIS
LIN {X 0.226,Y -612.654,Z 682.594,A 0.000,B 0.000,C 90.000,E1 322.924} C_DIS
LIN {X 0.290,Y -617.567,Z 682.591,A 0.000,B 0.000,C 90.000,E1 322.271} C_DIS
LIN {X 0.208,Y -624.834,Z 682.585,A 0.000,B 0.000,C 90.000,E1 321.251} C_DIS
LIN {X -0.136,Y -629.880,Z 682.581,A 0.000,B 0.000,C 90.000,E1 320.517} C_DIS
LIN {X 0.343,Y -636.166,Z 682.575,A 0.000,B 0.000,C 90.000,E1 319.461} C_DIS
LIN {X 0.028,Y -641.410,Z 682.570,A 0.000,B 0.000,C 90.000,E1 318.609} C_DIS
LIN {X 0.178,Y -647.818,Z 682.564,A 0.000,B 0.000,C 90.000,E1 317.472} C_DIS
LIN {X -0.009,Y -652.514,Z 682.559,A 0.000,B 0.000,C 90.000,E1 316.620} C_DIS
LIN {X 0.305,Y -656.918,Z 682.554,A 0.000,B 0.000,C 90.000,E1 315.729} C_DIS
LIN {X 0.195,Y -661.530,Z 682.549,A 0.000,B 0.000,C 90.000,E1 314.757} C_DIS
LIN {X 0.149,Y -664.803,Z 682.545,A 0.000,B 0.000,C 90.000,E1 314.028} C_DIS
LIN {X -0.323,Y -670.083,Z 682.538,A 0.000,B 0.000,C 90.000,E1 312.852} C_DIS
LIN {X 0.218,Y -674.168,Z 682.533,A 0.000,B 0.000,C 90.000,E1 311.838} C_DIS
LIN {X -0.144,Y -678.008,Z 682.527,A 0.000,B 0.000,C 90.000,E1 310.906} C_DIS
LIN {X 0.018,Y -680.673,Z 682.523,A 0.000,B 0.000,C 90.000,E1 310.172} C_DIS
LIN {X 0.213,Y -683.134,Z 682.519,A 0.000,B 0.000,C 90.000,E1 309.439} C_DIS
LIN {X -0.058,Y -686.065,Z 682.514,A 0.000,B 0.000,C 90.000,E1 308.508} C_DIS
LIN {X 0.353,Y -688.715,Z 682.509,A 0.000,B 0.000,C 90.000,E1 307.523} C_DIS
LIN {X 0.259,Y -691.065,Z 682.503,A 0.000,B 0.000,C 90.000,E1 306.583} C_DIS
LIN {X 0.141,Y -692.673,Z 682.499,A 0.000,B 0.000,C 90.000,E1 305.884} C_DIS
LIN {X -0.266,Y -695.038,Z 682.493,A 0.000,B 0.000,C 90.000,E1 304.739} C_DIS
LIN {X 0.228,Y -696.288,Z 682.489,A 0.000,B 0.000,C 90.000,E1 303.992} C_DIS
LIN {X 0.056,Y -698.086,Z 682.482,A 0.000,B 0.000,C 90.000,E1 302.832} C_DIS
LIN {X -0.088,Y -699.545,Z 682.476,A 0.000,B 0.000,C 90.000,E1 301.671} C_DIS
LIN {X 0.454,Y -700.401,Z 682.472,A 0.000,B 0.000,C 90.000,E1 300.924} C_DIS
LIN {X 0.241,Y -701.554,Z 682.464,A 0.000,B 0.000,C 90.000,E1 299.539} C_DIS
LIN {X 0.112,Y -702.145,Z 682.459,A 0.000,B 0.000,C 90.000,E1 298.615} C_DIS
LIN {X 0.155,Y -703.335,Z 682.449,A 0.000,B 0.000,C 90.000,E1 296.744} C_DIS
LIN {X -0.284,Y -704.011,Z 682.444,A 0.000,B 0.000,C 90.000,E1 295.848} C_DIS
LIN {X 0.000,Y -704.100,Z 682.442,A 0.000,B 0.000,C 90.000,E1 295.591} C_DIS
LIN {X -0.367,Y -703.838,Z 682.440,A 0.000,B 0.000,C 90.000,E1 295.155} C_DIS
LIN {X -0.082,Y -703.418,Z 682.438,A 0.000,B 0.000,C 90.000,E1 294.899} C_DIS
LIN {X -0.448,Y -701.835,Z 682.436,A 0.000,B 0.000,C 90.000,E1 294.463} C_DIS
LIN {X -0.309,Y -701.311,Z 682.435,A 0.000,B 0.000,C 90.000,E1 294.335} C_DIS
LIN {X -0.170,Y -700.506,Z 682.434,A 0.000,B 0.000,C 90.000,E1 294.207} C_DIS
LIN {X 0.176,Y -695.714,Z 682.432,A 0.000,B 0.000,C 90.000,E1 293.718} C_DIS
LIN {X -0.293,Y -694.228,Z 682.431,A 0.000,B 0.000,C 90.000,E1 293.643} C_DIS
LIN {X -0.126,Y -691.752,Z 682.431,A 0.000,B 0.000,C 90.000,E1 293.515} C_DIS
LIN {X 0.258,Y -687.423,Z 682.430,A 0.000,B 0.000,C 90.000,E1 293.334} C_DIS
LIN {X -0.022,Y -680.748,Z 682.429,A 0.000,B 0.000,C 90.000,E1 293.206} C_DIS
LIN {X 0.138,Y -678.628,Z 682.429,A 0.000,B 0.000,C 90.000,E1 293.153} C_DIS
LIN {X 0.170,Y -661.987,Z 682.428,A 0.000,B 0.000,C 90.000,E1 292.950} C_DIS
LIN {X -0.087,Y -651.543,Z 682.427,A 0.000,B 0.000,C 90.000,E1 292.823} C_DIS
LIN {X -0.193,Y -638.365,Z 682.425,A 0.000,B 0.000,C 90.000,E1 292.589} C_DIS
LIN {X 0.210,Y -628.289,Z 682.424,A 0.000,B 0.000,C 90.000,E1 292.333} C_DIS
LIN {X 0.056,Y -618.487,Z 682.423,A 0.000,B 0.000,C 90.000,E1 292.099} C_DIS
LIN {X 0.004,Y -594.528,Z 682.419,A 0.000,B 0.000,C 90.000,E1 291.408} C_DIS
LIN {X 0.148,Y -575.115,Z 682.416,A 0.000,B 0.000,C 90.000,E1 290.791} C_DIS
LIN {X 0.162,Y -562.658,Z 682.414,A 0.000,B 0.000,C 90.000,E1 290.429} C_DIS
LIN {X 0.080,Y -557.048,Z 682.412,A 0.000,B 0.000,C 90.000,E1 290.174} C_DIS
LIN {X 0.178,Y -555.475,Z 682.411,A 0.000,B 0.000,C 90.000,E1 289.993} C_DIS
LIN {X 0.136,Y -555.442,Z 682.411,A 0.000,B 0.000,C 90.000,E1 289.993} C_DIS
LIN {X 0.309,Y -554.604,Z 682.409,A 0.000,B 0.000,C 90.000,E1 289.631} C_DIS
LIN {X 0.050,Y -554.182,Z 682.405,A 0.000,B 0.000,C 90.000,E1 288.960} C_DIS
LIN {X -0.127,Y -553.793,Z 682.398,A 0.000,B 0.000,C 90.000,E1 287.583} C_DIS
LIN {X -0.038,Y -553.303,Z 682.388,A 0.000,B 0.000,C 90.000,E1 285.898} C_DIS
LIN {X 0.153,Y -552.790,Z 682.381,A 0.000,B 0.000,C 90.000,E1 284.481} C_DIS
LIN {X -0.197,Y -552.157,Z 682.373,A 0.000,B 0.000,C 90.000,E1 283.119} C_DIS
LIN {X -0.146,Y -551.428,Z 682.365,A 0.000,B 0.000,C 90.000,E1 281.715} C_DIS
LIN {X -0.224,Y -550.898,Z 682.359,A 0.000,B 0.000,C 90.000,E1 280.602} C_DIS
LIN {X -0.052,Y -549.931,Z 682.346,A 0.000,B 0.000,C 90.000,E1 278.341} C_DIS
LIN {X -0.013,Y -549.493,Z 682.335,A 0.000,B 0.000,C 90.000,E1 276.372} C_DIS
LIN {X -0.157,Y -549.248,Z 682.326,A 0.000,B 0.000,C 90.000,E1 274.702} C_DIS
LIN {X 0.114,Y -549.177,Z 682.318,A 0.000,B 0.000,C 90.000,E1 273.269} C_DIS
LIN {X -0.153,Y -548.929,Z 682.310,A 0.000,B 0.000,C 90.000,E1 271.892} C_DIS
LIN {X 0.117,Y -548.344,Z 682.303,A 0.000,B 0.000,C 90.000,E1 270.458} C_DIS
LIN {X -0.138,Y -547.359,Z 682.293,A 0.000,B 0.000,C 90.000,E1 268.797} C_DIS
LIN {X 0.140,Y -546.384,Z 682.284,A 0.000,B 0.000,C 90.000,E1 267.078} C_DIS
LIN {X -0.225,Y -545.603,Z 682.278,A 0.000,B 0.000,C 90.000,E1 265.988} C_DIS
LIN {X 0.060,Y -544.556,Z 682.270,A 0.000,B 0.000,C 90.000,E1 264.546} C_DIS
LIN {X 0.261,Y -543.678,Z 682.263,A 0.000,B 0.000,C 90.000,E1 263.394} C_DIS
LIN {X -0.017,Y -542.180,Z 682.256,A 0.000,B 0.000,C 90.000,E1 262.008} C_DIS
LIN {X 0.038,Y -539.403,Z 682.240,A 0.000,B 0.000,C 90.000,E1 259.162} C_DIS
LIN {X -0.071,Y -537.933,Z 682.230,A 0.000,B 0.000,C 90.000,E1 257.465} C_DIS
LIN {X -0.092,Y -536.518,Z 682.221,A 0.000,B 0.000,C 90.000,E1 255.755} C_DIS
LIN {X 0.264,Y -535.503,Z 682.214,A 0.000,B 0.000,C 90.000,E1 254.574} C_DIS
LIN {X -0.005,Y -533.439,Z 682.203,A 0.000,B 0.000,C 90.000,E1 252.598} C_DIS
LIN {X 0.034,Y -531.160,Z 682.191,A 0.000,B 0.000,C 90.000,E1 250.296} C_DIS
LIN {X 0.116,Y -529.369,Z 682.183,A 0.000,B 0.000,C 90.000,E1 248.847} C_DIS
LIN {X -0.131,Y -527.729,Z 682.176,A 0.000,B 0.000,C 90.000,E1 247.720} C_DIS
LIN {X 0.267,Y -525.630,Z 682.168,A 0.000,B 0.000,C 90.000,E1 246.230} C_DIS
LIN {X -0.181,Y -522.695,Z 682.158,A 0.000,B 0.000,C 90.000,E1 244.537} C_DIS
LIN {X 0.030,Y -521.133,Z 682.154,A 0.000,B 0.000,C 90.000,E1 243.640} C_DIS
LIN {X 0.060,Y -517.117,Z 682.142,A 0.000,B 0.000,C 90.000,E1 241.591} C_DIS
LIN {X 0.104,Y -514.738,Z 682.136,A 0.000,B 0.000,C 90.000,E1 240.411} C_DIS
LIN {X 0.265,Y -510.313,Z 682.124,A 0.000,B 0.000,C 90.000,E1 238.329} C_DIS
LIN {X 0.138,Y -508.345,Z 682.119,A 0.000,B 0.000,C 90.000,E1 237.454} C_DIS
LIN {X -0.221,Y -504.980,Z 682.111,A 0.000,B 0.000,C 90.000,E1 236.008} C_DIS
LIN {X 0.173,Y -502.191,Z 682.104,A 0.000,B 0.000,C 90.000,E1 234.769} C_DIS
LIN {X -0.016,Y -498.550,Z 682.096,A 0.000,B 0.000,C 90.000,E1 233.290} C_DIS
LIN {X 0.189,Y -494.121,Z 682.086,A 0.000,B 0.000,C 90.000,E1 231.457} C_DIS
LIN {X -0.079,Y -489.698,Z 682.076,A 0.000,B 0.000,C 90.000,E1 229.666} C_DIS
LIN {X 0.023,Y -484.659,Z 682.064,A 0.000,B 0.000,C 90.000,E1 227.514} C_DIS
LIN {X 0.054,Y -481.022,Z 682.055,A 0.000,B 0.000,C 90.000,E1 225.972} C_DIS
LIN {X -0.120,Y -478.195,Z 682.049,A 0.000,B 0.000,C 90.000,E1 224.757} C_DIS
LIN {X -0.003,Y -473.138,Z 682.037,A 0.000,B 0.000,C 90.000,E1 222.567} C_DIS
